// TwinCAT 3 PLC project Hammerschmied
// ProgramVersion: 3.1.4023.0
// libraries:
//   EfficientIO Communicator, * (EfficientIO)
//   EfficientIO Energy Basic, * (EfficientIO)
//   EfficientIO ModbusTCP, * (EfficientIO)
//   Lynus Persistent Data V1, * (Lynus AG)
//   Lynus Standards, * (EfficientIO)
//   Tc2_Standard, * (Beckhoff Automation GmbH)
//   Tc2_System, * (Beckhoff Automation GmbH)
//   Tc2_Utilities, * (Beckhoff Automation GmbH)
//   Tc3_Module, * (Beckhoff Automation GmbH)
// project tree:
//   / FastTask.TcTTO (not stored), MiddleTask.TcTTO, SlowTask.TcTTO
//   FB/ FB_EMS_T.TcPOU (excluded from build), FB_EMS_V12.TcPOU, FB_EM_Beckhoff_KL3403.TcPOU (not stored), FB_IntervalBit.TcPOU (not stored)
//   POUs/ prgBattery.TcPOU, prgComEffIO.TcPOU, prgCS.TcPOU, prgEM.TcPOU, prgEMS.TcPOU, prgGrid.TcPOU, prgHouse.TcPOU, prgPersistent.TcPOU (not stored), prgPV.TcPOU, prgRWEffIO.TcPOU, prgVarEffIO.TcPOU (not stored)
// real-time tasks:
//   TASK FastTask: cycle T#5ms, priority 6, ADS port 350
//   TASK MiddleTask: cycle T#10ms, priority 8, ADS port 351
//   TASK SlowTask: cycle T#20ms, priority 10, ADS port 352
// I/O:
//   DEVICE Gerät 2 (CX-BK)
//     Box 1 (CX-BK)
// variable links:
//   Hammerschmied/Hammerschmied Instance <-> Device 2 (CX-BK)/Box 1 (CX-BK)
//     MiddleTask Inputs/prgEM.fbEM1.fbKL3403.byStateCH1 <-> Term 2 (KL3403)/Channel 1/Status
//     MiddleTask Inputs/prgEM.fbEM1.fbKL3403.byStateCH2 <-> Term 2 (KL3403)/Channel 2/Status
//     MiddleTask Inputs/prgEM.fbEM1.fbKL3403.byStateCH3 <-> Term 2 (KL3403)/Channel 3/Status
//     MiddleTask Inputs/prgEM.fbEM1.fbKL3403.iDataInCH1 <-> Term 2 (KL3403)/Channel 1/Daten Ein
//     MiddleTask Inputs/prgEM.fbEM1.fbKL3403.iDataInCH2 <-> Term 2 (KL3403)/Channel 2/Daten Ein
//     MiddleTask Inputs/prgEM.fbEM1.fbKL3403.iDataInCH3 <-> Term 2 (KL3403)/Channel 3/Daten Ein
//     MiddleTask Inputs/prgEM.fbKBusState.uiKBusState_OUT <-> Inputs/State
//     MiddleTask Outputs/prgEM.fbEM1.fbKL3403.byCntrCH1 <-> Term 2 (KL3403)/Channel 1/Kontrolle
//     MiddleTask Outputs/prgEM.fbEM1.fbKL3403.byCntrCH2 <-> Term 2 (KL3403)/Channel 2/Kontrolle
//     MiddleTask Outputs/prgEM.fbEM1.fbKL3403.byCntrCH3 <-> Term 2 (KL3403)/Channel 3/Kontrolle

CONFIGURATION Hammerschmied
    RESOURCE PLC ON TwinCAT3
        TASK MiddleTask(INTERVAL := T#10ms, PRIORITY := 8);
        TASK SlowTask(INTERVAL := T#20ms, PRIORITY := 10);
        PROGRAM prgBattery WITH MiddleTask : prgBattery;
        PROGRAM prgCS WITH MiddleTask : prgCS;
        PROGRAM prgEMS WITH MiddleTask : prgEMS;
        PROGRAM prgGrid WITH MiddleTask : prgGrid;
        PROGRAM prgHouse WITH MiddleTask : prgHouse;
        PROGRAM prgPersistent WITH MiddleTask : prgPersistent;
        PROGRAM prgPV WITH MiddleTask : prgPV;
        PROGRAM prgEM WITH MiddleTask : prgEM;
        PROGRAM prgComEffIO WITH SlowTask : prgComEffIO;
    END_RESOURCE
END_CONFIGURATION

// ---- POUs/prgBattery.TcPOU
PROGRAM prgBattery
VAR PERSISTENT
	bEnableBattery				: BOOL;							//{#lynus.ag#()}
	byPrioBattery				: BYTE;							//{#lynus.ag#()}
	lrMaxCapacityBattery		: LREAL;						//{#lynus.ag#()}
	lrCounterBattProd			: LREAL;						//{#lynus.ag#()}
	lrCounterBattCons			: LREAL;						//{#lynus.ag#()}
	by_Min_BatterySOC			: BYTE;							//{#lynus.ag#()}
	by_Max_BatterySOC			: BYTE;							//{#lynus.ag#()}
END_VAR
VAR
	fbBattery					: FB_Xelectrix_Powerbox_v2_2;
	fbBattCounter				: FB_EnergyCounter;
	bIsEnabledBattery			: BOOL;							//{#lynus.ag#()}
	bResetBattery				: BOOL;							//{#lynus.ag#()}
	bSResetBattery				: BOOL;							//{#lynus.ag#()}
	byErrorWarningBattery		: BYTE;							//{#lynus.ag#()}
	dwSOCBattery				: DWORD;						//{#lynus.ag#()}
	rTargetPowerBattery			: REAL;							//{#lynus.ag#()}
	lrPowerBattery				: LREAL;						//{#lynus.ag#()}
	lrActualCapacityBattery		: LREAL;						//{#lynus.ag#()}
	mtest: BOOL;

	int_GridState: INT;											//{#lynus.ag#()}
	int_BatteryState: INT;										//{#lynus.ag#()}
	int_OperatingState: INT;									//{#lynus.ag#()}
	int_ErrorState: INT;										//{#lynus.ag#()}

	FB_Interval: FB_IntervalBit;
	m_IslandOperationStart: BOOL;								//{#lynus.ag#()}
	m_IslandOperationOngoing: BOOL;								//{#lynus.ag#()}
	m_IslandOperationStop: BOOL;								//{#lynus.ag#()}
	t_Interval :TIME:=T#30M;
	t_HightTime :TIME:=T#1S;
	
	m_BatteryErrorActive: BOOL;									//{#lynus.ag#()}
	m_BatteryModbusCommError: BOOL;								//{#lynus.ag#()}
	m_BatteryTargetSPError: BOOL;								//{#lynus.ag#()}
	Ton_Delay_BatteryError: Ton;
	Ton_Delay_BatteryModbusError: Ton;
	Ton_Delay_BatterySPError: Ton;	
	by_S_Min_BatterySOC			: BYTE;							//{#lynus.ag#()}
	by_S_Max_BatterySOC			: BYTE;							//{#lynus.ag#()}
	
END_VAR


IF mtest THEN
	Lynus_Standards.GVL_Energy.stDataOfBatteryInverters[1,1].rTargetPowerEMS:=0;
	mtest:=FALSE;
 END_IF
 
 
 
fbBattery(
	bEnable:= bEnableBattery, 
	bActivateControl:= TRUE, 
	byUnitID:= 1, 
	byPriority:= byPrioBattery, 
	diNrOfEMS_IN:= prgEMS.fbEMS.diNrOfEMS_OUT, 
	lrMaxCapacityBattery:= lrMaxCapacityBattery, 
	sIPAdress:= '192.168.1.235', 						// modify IP Adress
	bReset:= bResetBattery, 
	by_minDischargeSOC := by_Min_BatterySOC,
	by_maxChargeSOC := by_Max_BatterySOC,
	stDataXelectrix=> , 
	stDataBatt=> , 
	stDataBattInverter=> , 
	stDataEMPower_Grid=> , 
	stDataEMCounter_Grid=> , 
	diNrOfBatt_OUT=> , 
	diNrOfBattInverter_OUT=> , 
	diNrOfEM_OUT_Grid=> , 
	lrMaxCapacityBattery_OUT=> ,	
	by_SminDischargeSOC	=> by_S_Min_BatterySOC,	
	by_SmaxChargeSOC=> by_S_Max_BatterySOC
);
	
//Out
bIsEnabledBattery := fbBattery.stDataBatt.bEnabled;
	bSResetBattery := fbBattery.stDataBattInverter.bStateReset;
		dwSOCBattery := fbBattery.stDataBatt.dwSOC;
			rTargetPowerBattery := fbBattery.stDataBattInverter.rTargetPower;
				lrPowerBattery := fbBattery.stDataBatt.lrPower;
					lrActualCapacityBattery := fbBattery.lrMaxCapacityBattery_OUT;	
						byErrorWarningBattery := fbBattery.stDataBatt.byErrorWarning;
						
						
// EnergyCounter
fbBattCounter(
	byActiveTariff:= 1, 
	lrPowerInput:= lrPowerBattery, 
	lrTotalCounterEnergy_Consumption=> , 
	lrTotalCounterEnergy_Production=> , 
	lrCounterEnergyT1_Consumption=> , 
	lrCounterEnergyT2_Consumption=> , 
	lrCounterEnergyT1_Production=> , 
	lrCounterEnergyT2_Production=> );
	
IF fbBattCounter.lrTotalCounterEnergy_Production > lrCounterBattProd THEN  	
	lrCounterBattProd := fbBattCounter.lrTotalCounterEnergy_Production;
END_IF

IF fbBattCounter.lrTotalCounterEnergy_Consumption > lrCounterBattCons THEN  	
	lrCounterBattCons := fbBattCounter.lrTotalCounterEnergy_Consumption;
END_IF

// send e states to cloud
int_GridState 		:= fbBattery.stDataXelectrix.eGridState;
int_BatteryState	:= fbBattery.stDataXelectrix.eBatteryState;
int_OperatingState	:= fbBattery.stDataXelectrix.eOperatingState;
int_ErrorState		:= fbBattery.stDataXelectrix.eErrorState;


// create bits when battery is in island operation

FB_Interval(
	m_Input			:=  prgBattery.fbBattery.stDataXelectrix.eGridState = 2,	//   2 = Island Mode 
	t_Interval 		:= t_Interval , 
	t_HighTime		:= t_HightTime, 
	m_RisingEdge	=> m_IslandOperationStart, 
	m_Interval		=> m_IslandOperationOngoing, 
	m_FallingEdge	=> m_IslandOperationStop);

// monitoring Battery status

Ton_Delay_BatteryError (In := fbBattery.stDataXelectrix.eErrorState =2,
						PT :=T#5S,
						Q => m_BatteryErrorActive);

Ton_Delay_BatteryModbusError (	In := fbBattery.stDataXelectrix.eErrorState = 1,
								PT :=T#10M,
								Q => m_BatteryModbusCommError);						

Ton_Delay_BatterySPError (	In := ABS(fbBattery.iSetpointPower/10-lrPowerBattery) > 20 AND fbBattery.stDataXelectrix.eGridState<>2 AND fbBattery.stDataBatt.dwSOC<90,	// not alarming during island operation
							PT :=T#1M,
							Q => m_BatteryTargetSPError);

END_PROGRAM

// ---- POUs/prgEMS.TcPOU
PROGRAM prgEMS
VAR PERSISTENT
	byMaxDepthOfDischrgEPO		: BYTE;							//{#lynus.ag#()}
	byPrioMinChrgBattSOCInEPO	: BYTE;							//{#lynus.ag#()}
	byResChrgfromGridToBatt		: BYTE;							//{#lynus.ag#()}
	byReserveSOCEPO				: BYTE;							//{#lynus.ag#()}
	uiUpdateTime				: UINT;							//{#lynus.ag#()}
	bEnableEMS					: BOOL;							//{#lynus.ag#()}
	bAllowChrgFromGrid			: BOOL;							//{#lynus.ag#()}
	rMainFuseCSEMS				: REAL;							//{#lynus.ag#()}
	iOperationModeEMS			: INT;							//{#lynus.ag#()}
	by_MinSOC_AdaptiveLC		: BYTE;							//{#lynus.ag#()}
END_VAR
VAR
	fbEMS						: FB_EMS_V12;
	bIsEnableEMS				: BOOL;							//{#lynus.ag#()}
	bStateAllowChrgFromGrid		: BOOL;							//{#lynus.ag#()}
	bHPActivate					: BOOL;							//{#lynus.ag#()}
	bControllingState			: BOOL;							//{#lynus.ag#()}
	iMessageEMS					: INT;							//{#lynus.ag#()}
	rHeartbeatEMS				: REAL;							//{#lynus.ag#()}
	rErrorWarningEMS			: REAL;							//{#lynus.ag#()}
	rReadyEMS					: REAL;							//{#lynus.ag#()}
	rNewBatteryPowerEMS			: REAL;							//{#lynus.ag#()}
	b_EnableBatteryChargingControl				: BOOL:=TRUE;							//{#lynus.ag#()}
	b_StartReleaseBatteryCharging				: BOOL;									//{#lynus.ag#()}
	b_StopReleaseBatteryCharging				: BOOL;									//{#lynus.ag#()}
	b_TimeBasedReleaseChargingBattery			: BOOL;									//{#lynus.ag#()}
	b_StartManualCharging						: BOOL;									//{#lynus.ag#()}
	b_StartManualCharging_SOC					: BOOL;									//{#lynus.ag#()}
	r_Charging_SOC_SetPoint						: REAL;									//{#lynus.ag#()}
	RS_ManualCharging: Rs;
	RS_ManualCharging_SOC: Rs;
	TON_ManualCharging: Ton;
	time_ManualCharging: TIME:=T#2H;
	r_trig_ManualCharging: R_trig;
	f_trig_ManualCharging: f_trig;
	r_trig_ManualCharging_SOC: R_trig;
	f_trig_ManualCharging_SOC: f_trig;
	r_trig_b_StartManualCharging: R_trig;
	r_trig_b_StartManualCharging_SOC: R_trig;
	m_test: BOOL;
	b_dummy						: bool;									//{#lynus.ag#()}
	iOperationModeEMS_actual			: INT;							//{#lynus.ag#()}

	mtest: BOOL;
	m_Enable_Dynamic_LM: BOOL;
END_VAR

fbEMS.stSetupEMS.bAllowChrgFromGrid := bAllowChrgFromGrid or RS_ManualCharging.Q1;
fbEMS.stSetupEMS.byMaxDepthOfDischrgEPO := byMaxDepthOfDischrgEPO;
fbEMS.stSetupEMS.byPrioMinChrgBattSOCInEPO := byPrioMinChrgBattSOCInEPO;
fbEMS.stSetupEMS.byResChrgfromGridToBatt := byResChrgfromGridToBatt;
fbEMS.stSetupEMS.byReserveSOCEPO := byReserveSOCEPO;
fbEMS.stSetupEMS.rSizeMainFuseCS := rMainFuseCSEMS;
fbEMS.stSetupEMS.uiUpdateTime := uiUpdateTime;
(*IF m_Enable_Dynamic_LM THEN
	IF prgBattery.dwSOCBattery > byMinSOCdynamicLM AND NOT prgCS.bCarConnected THEN
		iOperationModeEMS := 1;
	ELSE
		iOperationModeEMS := 3;
	END_IF  
END_IF

IF iOperationModeEMS = 0 THEN fbEMS.eOperationMode := E_OperatingMode_EMS.eAllOff;
ELSIF iOperationModeEMS = 1 THEN fbEMS.eOperationMode := E_OperatingMode_EMS.eSelfConsumption;	
ELSIF iOperationModeEMS = 2 THEN fbEMS.eOperationMode := E_OperatingMode_EMS.ePeakLoadCapping;
ELSIF iOperationModeEMS = 3 THEN fbEMS.eOperationMode := E_OperatingMode_EMS.eLoadManagement;			
END_IF
*)
IF iOperationModeEMS = 0 THEN 
	fbEMS.eOperationMode_Ext := E_OperatingMode_EMS.eAllOff;
ELSIF iOperationModeEMS = 1 THEN 
	fbEMS.eOperationMode_Ext := E_OperatingMode_EMS.eSelfConsumption;	
ELSIF iOperationModeEMS = 2 THEN 
	fbEMS.eOperationMode_Ext := E_OperatingMode_EMS.ePeakLoadCapping;
ELSIF iOperationModeEMS = 3 THEN 
	fbEMS.eOperationMode_Ext := E_OperatingMode_EMS.eLoadManagement;			
ELSIF iOperationModeEMS = 4 THEN 
	fbEMS.eOperationMode_Ext := E_OperatingMode_EMS.eAdaptiveLoadControl;		
END_IF

fbEMS(
	bEnable:= bEnableEMS, 
	diNrOfEM_IN_ECS:= , 
	stSetupEMS:= , 
	eOperationMode_Ext:= , 
	eSpeedModeBackendController:= E_SpeedModeBackendController_EMS.eSlow,	//.efast, 
	eSpeedModeLocalController:= E_SpeedModeLocalController_EMS.eSlow,    //efast,
	bZeroPowerRegulation	:= FALSE, 
	b_EnableBatteryChargingControl	:= b_EnableBatteryChargingControl,
	b_StartReleaseBatteryCharging 	:= b_StartReleaseBatteryCharging OR r_trig_ManualCharging.Q ,
	b_StopReleaseBatteryCharging 	:= b_StopReleaseBatteryCharging OR (f_trig_ManualCharging.Q AND NOT b_StartReleaseBatteryCharging) OR (f_trig_ManualCharging_SOC.Q AND NOT b_StartReleaseBatteryCharging) ,
	by_MinSOC_AdaptiveLC:= by_MinSOC_AdaptiveLC, 
	bActivateHP:= bHPActivate, 
	bControllingState:= TRUE, //bControllingState, 
	rHeartbeat:= rHeartbeatEMS, 
	rErrorWarning:= rErrorWarningEMS, 
	rEnergyOptReady:= rReadyEMS, 
	rNewBattPower:= rNewBatteryPowerEMS,
	b_AnyCarConnected:= prgCS.bCarConnected , 
	rMaxBattChargingPower:= , 
	rPeakDetectionforCalculation:= , 
	eMessageEMS=> iMessageEMS, 
	bStateEnable=> bIsEnableEMS, 
	bStateAllowChrgFromGrid=> bStateAllowChrgFromGrid, 
	bMissingPowerData=> , 
	bSurplusAvailable=> , 
	byProgress=> , 
	uiState_OUT=> , 
	diNrOfEMS_OUT=> , 
	arrMinPrioReached=> , 
	arrMaxPrioReached=> , 
	b_TimeBasedReleaseChargingBattery => b_TimeBasedReleaseChargingBattery);

iOperationModeEMS_actual := fbEMS.eOperationMode;

(*
fbEMS(
	bEnable:= bEnableEMS, 
	diNrOfEM_IN_ECS:= , 
	stSetupEMS:= , 
	eOperationMode:= , 
	eSpeedModeBackendController:= E_SpeedModeBackendController_EMS.efast, 
	eSpeedModeLocalController:= E_SpeedModeLocalController_EMS.efast,
	bActivateHP:= bHPActivate, 
	bControllingState:= TRUE, //bControllingState, 
	rHeartbeat:= rHeartbeatEMS, 
	rErrorWarning:= rErrorWarningEMS, 
	rEnergyOptReady:= rReadyEMS, 
	rNewBattPower:= rNewBatteryPowerEMS, 
	b_ZeroPowerRegulation	:= FALSE,
	b_EnableBatteryChargingControl	:= b_EnableBatteryChargingControl,
	b_StartReleaseBatteryCharging 	:= b_StartReleaseBatteryCharging OR r_trig_ManualCharging.Q ,
	b_StopReleaseBatteryCharging 	:= b_StopReleaseBatteryCharging OR (f_trig_ManualCharging.Q AND NOT b_StartReleaseBatteryCharging) OR (f_trig_ManualCharging_SOC.Q AND NOT b_StartReleaseBatteryCharging) ,
	rMaxBattChargingPower			:= ,
	rPeakDetectionforCalculation	:=,
	eMessageEMS=> iMessageEMS, 
	bStateEnable=> bIsEnableEMS, 
	bStateAllowChrgFromGrid=> bStateAllowChrgFromGrid, 
	bMissingPowerData=> , 
	bSurplusAvailable=> , 
	byProgress=> , 
	uiState_OUT=> , 
	diNrOfEMS_OUT=> , 
	arrMinPrioReached=> , 
	arrMaxPrioReached=> ,
	b_TimeBasedReleaseChargingBattery => b_TimeBasedReleaseChargingBattery);
*)
	
// code for manual charging button, time hardcoded to 2h with variable 	time_ManualCharging
	
r_trig_b_StartManualCharging(clk:=b_StartManualCharging);
r_trig_b_StartManualCharging_SOC(clk:=b_StartManualCharging_SOC);
RS_ManualCharging_SOC(	Set := r_trig_b_StartManualCharging_SOC.Q AND NOT RS_ManualCharging_SOC.Q1 AND REAL_TO_DWORD(r_Charging_SOC_SetPoint) > prgBattery.dwSOCBattery AND NOT b_TimeBasedReleaseChargingBattery AND NOT RS_ManualCharging.Q1,
						Reset1 := (r_trig_b_StartManualCharging_SOC.Q AND RS_ManualCharging_SOC.Q1) OR REAL_TO_DWORD(r_Charging_SOC_SetPoint) <= prgBattery.dwSOCBattery OR b_StartReleaseBatteryCharging);
IF 	(r_trig_b_StartManualCharging.Q OR r_trig_b_StartManualCharging_SOC.Q) AND NOT b_TimeBasedReleaseChargingBattery AND NOT RS_ManualCharging.Q1 THEN
	RS_ManualCharging.SET:=TRUE;
ELSIF (r_trig_b_StartManualCharging.Q  AND RS_ManualCharging.Q1) OR (TON_ManualCharging.Q AND NOT RS_ManualCharging_SOC.Q1)  OR b_StartReleaseBatteryCharging OR f_trig_ManualCharging_SOC.Q THEN
	RS_ManualCharging.RESET1:=TRUE;		
END_IF
TON_ManualCharging(	In:=RS_ManualCharging.Q1, PT:= time_ManualCharging);

RS_ManualCharging();
RS_ManualCharging.SET:=FALSE;
RS_ManualCharging.RESET1:=FALSE;
r_trig_ManualCharging(clk:=RS_ManualCharging.Q1);
f_trig_ManualCharging(clk:=RS_ManualCharging.Q1);
r_trig_ManualCharging_SOC(clk:=RS_ManualCharging_SOC.Q1);
f_trig_ManualCharging_SOC(clk:=RS_ManualCharging_SOC.Q1);

			
// Test
IF REAL_TO_DWORD(r_Charging_SOC_SetPoint) > prgBattery.dwSOCBattery  THEN
	mtest := TRUE;
ELSE
	mtest := FALSE;
END_IF

END_PROGRAM

// ---- FB/FB_EMS_V12.TcPOU
FUNCTION_BLOCK FB_EMS_V12
VAR_INPUT PERSISTENT
	bEnable										: BOOL;																								//{#lynus.ag#()} //Enable and dissable this function
	diNrOfEM_IN_ECS								: DINT;																								//Number of the electric meter for incoming power data. (Its for the complete consumption of all charging stations)
	stSetupEMS									: ST_Setup_EMS := (uiUpdateTime := 15);																//{#lynus.ag#()} //Setup EMS
	eOperationMode_Ext							: E_OperatingMode_EMS;																				//{#lynus.ag#()} //Operation Mode EMS
	eSpeedModeBackendController					: E_SpeedModeBackendController_EMS;																	//Speed for the Controller what discharge the Battery when the commands come from the Backend
	eSpeedModeLocalController					: E_SpeedModeLocalController_EMS;																	//Speed for the local Controller for charge and discharge the Battery
	bZeroPowerRegulation						: BOOL;																								//{#lynus.ag#()} // activates the Battery discharging before using the mains during LoadManagement; Line 1728/1732/1738
	b_EnableBatteryChargingControl				: BOOL;																								//{#lynus.ag#()} //  
	b_StartReleaseBatteryCharging				: BOOL;																								//{#lynus.ag#()} //  
	b_StopReleaseBatteryCharging				: BOOL;																								//{#lynus.ag#()} //  
	by_MinSOC_AdaptiveLC						: BYTE; 
END_VAR
VAR_INPUT
	bActivateHP									: BOOL;																								//{#lynus.ag#()} //Activate the Heating pumps when the Backend deliver the signal. NOT OVERRIDE
	bControllingState							: BOOL;																								//{#lynus.ag#()} //The control state of the service is linked here. NOT OVERRIDE
	rHeartbeat									: REAL;																								//{#lynus.ag#()} //Heartbeat from the Service. NOT OVERRIDE
	rErrorWarning								: REAL;																								//{#lynus.ag#()} //Error or Warning from the Service. NOT OVERRIDE
	rEnergyOptReady								: REAL;																								//{#lynus.ag#()} //Energy Optimization Service Ready. NOT OVERRIDE
	rNewBattPower								: REAL;																								//{#lynus.ag#()} //New Battery Power from Backend Service. NOT OVERRIDE
	b_AnyCarConnected							: BOOL;																								// requrired for the dadaptive load control 
	rMaxBattChargingPower						: REAL:=100;																								// Maximum Battery Charging power in percent
	rPeakDetectionforCalculation				: REAL:=3;																								// Value for Peak detection, was original 3 but caused issues with fast changing loads (e.g. industrie)
END_VAR
VAR_OUTPUT
	eMessageEMS									: Lynus_Standards.E_Message_EMS;																	//EMS Message
	bStateEnable								: BOOL;																								//{#lynus.ag#()} //Show if the ems function is enabled or not
	bStateAllowChrgFromGrid						: BOOL;																								//{#lynus.ag#()} //Show the State if the charging from grid is allowed or not
	bMissingPowerData							: BOOL;																								//Missing data on the max power setup from one ore more devices
	bSurplusAvailable							: BOOL;																								//Variable that indicates if there is surplus or not
	byProgress									: BYTE;																								//Shows the Progress from the new Calculation when we have Surplus. When we have no Surplus and we discharge the batterys this Value is on 100
	uiState_OUT									: UINT;																								//Actual State
	diNrOfEMS_OUT								: DINT;																								//Active Number from the EMS Function for using on other functions
	arrMinPrioReached							: ARRAY[1..5] OF BOOL;																				//Shows if all different devices types are set to 0% with the target power ([1] = Battery, [2] = HP, [3] = EHE, [4] = OBC, [5] = ECS)
	arrMaxPrioReached							: ARRAY[1..5] OF BOOL;																				//Shows if all different devices types are set to 100% with the target power ([1] = Battery, [2] = HP, [3] = EHE, [4] = OBC, [5] = ECS)	
	b_TimeBasedReleaseChargingBattery			: BOOL;																								//
END_VAR	
VAR
	eOperationMode								: E_OperatingMode_EMS;																				//{#lynus.ag#()} //Operation Mode EMS
	(*-----------------------------------------------------------------------Internal Variables and Functions for connection to the Backend--------------------------------------------------------------------------------*)
	fbPIDDischrgCmdFromBackend					: FB_PID;																							//PID Contrller what controll the discharging power from the Battery when the controlling from backend is activated
	timDissableFunctions						: TON;																								//Timer to dissable the Function after Lynus_Standards.Constants_General.tTimeDissableLynusFunctions Days without connection to the Lynus Cloud
	timResetConnectionOnGVL						: TON;																								//Timer to try reset the connection Flag on the GVL. (When somebody delete the Connection Function and make only a onlinechange)
	timHB										: TON;																								//Timer to check the Heartbeat from the Backendservice
	timPIDDischrgCmdFromBackend					: TON;																								//Timer to set the output from the pid controller to 0 due to internal control deviations (Backend Mode)
	timCorrectionSetpoint						: TOF;																								//Timer to make the correction on the Setpoint for Battery power. This is neccessary to give time to the inverter and Grid to adjust on the new values
	timErrorWarning								: TON;																								//Timer to enable the Function Backend Mode after a Error or Warning
	timEnergyOptReady							: TON;																								//Timer to enable the Function Backend Mode after the Backend Service is ready
	timControlingState							: TON;																								//Timer to enable the controlling over the Backend Mode
	timResetActivateHP							: TON;																								//Timer to reset the Activate HP Command from the Backend Service
	FPEnablePID									: R_TRIG;																							//Internal positive edge
	FPMakeCorrection							: R_TRIG;																							//Internal positive edge
	bDischrgCmdFromBackendOK					: BOOL;																								//Allowed to controll the Devices from Backend
	rHeartbeat_CP								: REAL;																								//Compare the Heartbeat from the Backend
	rControllerQPIDDischrgCmdFromBackend		: REAL;																								//Controller output from pid controll over Backend Mode
	rNewBattPower_CP							: REAL;																								//New Battery power to ckeck if we have received a new Value in kW
	lrActualPowerBatterys						: LREAL;																							//Actual Power from the Batterys in kW
	lrErrorPIDCorrectionDischrgCmdFromBackend	: LREAL;																							//Limit the Error on the pid controller for discahrge the battery on the controll over Backend Mode
	lrNewBatteryPowerWithCorrection				: LREAL;																							//The New Battery power from the Backend with correction that we dont insert power in the Grid
	liLPDischrgCmdFromBackend					: LINT;																								//Loop to send the command from Backend to the Devices
	(*-----------------------------------------------------------------------------------Rest of internal Variabels and Functions---------------------------------------------------------------------------------------*)
	fbMessagesEMS								: FB_EMS_Message;																					//FB to create the Messages for this Function
	fbNumberDevice								: FB_NumberOfDevice;																				//Function block to calcualte the number of the Device
	fbTaskIndex									: GETCURTASKINDEX;																					//Function to read out the Task Index in witch the function is running
	fbPIDBatterySC								: FB_PID;																							//PID Controller to discharge the battery in the self consumption mode
	fbPIDBatteryEPO								: FB_PID;																							//PID Controller to discharge the battery in the emergency power mode
	fbPIDBatteryPLCLM_Dischrg					: FB_PID;																							//PID Controller to Dischage the battery on load management mode and peak shaving mode
	fbPIDBatteryPLCLM_Chrg						: FB_PID;																							//PID Controller to Charge the battery on load management mode and peak shaving mode
	timCalculateNewPowerValue					: TON;																								//Timer to start a new session to calculate the new power value for the devices
	timPIDSC									: TON;																								//Timer to set the output from the pid controller to 0 due to internal control deviations (Self consumption mode)
	timPIDEPO									: TON;																								//Timer to set the output from the pid controller to 0 due to internal control deviations (Emergency power mode)
	timCorrectionECS							: TON;																								//Timer for make the correction for ECS in the Load management and peak capping mode with use the separate fuse
	timErrorGridMessurement						: TON;																								//Timer with delay to stop the EMS Function if we have a error on the Grid messurement
	timTimeout									: TON;																								//Timer for Timout
	timCutPeaks									: TOF;																								//Timer to cut peaks on the grid. The system waits for this time for strong and short peaks before regulating.
	timDelayStart								: TOF;																								//Timer with the delay to start the ems function after a online change
	timResetDisableECS							: TOF;																								//Timer to reset the dissbling the ECS after a Error from the Electric Meter what messure the power from all ECS
	FPEPO										: R_TRIG;																							//Internal positive edge
	FNEPO										: F_TRIG;																							//Internal negative edge
	eOperationModeEMS_CP						: E_OperatingMode_EMS;																				//Operation Mode EMS/Battery to compare with the original variable
	arrPD										: ARRAY[1..12] OF FB_PersistentData_Number;															//Function to save persistent data
	arrTimBatterysAreFull						: ARRAY[1..Constants_Energy.diMaxNumberOfBatteryInverters] OF TON;									//Timer start for each Battery when is full
	arrActualStepInTurn_CP						: ARRAY[1..2] OF BYTE;																				//Actual Step in turn to compare with original variable
	arrActualPrioInTurn							: ARRAY[1..5] OF BYTE;																				//Actual Priority (1-255) that is currently in turn ([1] = Battery, [2] = HP, [3] = EHE, [4] = OBC, [5] = ECS)
	arrActualStepInTurn							: ARRAY[1..2] OF BYTE;																				//Actual Step (1-10) from step switched devices that is currently in turn ([1] = HP, [2] = EHE)
	arrLPPrioZeroSetToZeroP						: ARRAY[1..5] OF LINT;																				//Array with loop to set each device with priority 0 to the target power value 
	arrCTCheckActivePrio						: ARRAY[1..5] OF LINT;																				//Array with loop to check the actual prioritys
	bEPMActive									: BOOL;																								//Emergency power mode is active
	bChargePrioBatterysOnEPO					: BOOL;																								//Load batterys that made a island grid first to the adjustable SOC before start with al other devices
	bStepWasOn100								: BOOL;																								//Its true when the actual step from step switched devices was on 100%
	bECSPrio255									: BOOL;																								//True when we reached the max prio of the charging stations
	bStopAll									: BOOL;																								//Stop the EMS when we some is happend what make trouble
	bDisableECS									: BOOL;																								//Dissable the ECS when the EM what messure the power from all ECS has a error
	bErrorOnGridMessurement						: BOOL;																								//Shows if on the Grid Messurement is a error and stop then the EMS Function
	bNoPowerForECS								: BOOL;																								//Variable what shows that we dont can give more power on the ECS because we have to much power on the Fuse line on wich the ECS is connected
	bySmGrActiveCommonPrio_CP					: BYTE;																								//Smalest or greatest active common priority of the devices to compare with the original varible
	byLPSmActiveCommonPrio						: BYTE;																								//Loop to check the smalest active common priority
	bySmGrActiveCommonPrio						: BYTE;																								//Smalest or greatest active common priority of the devices
	bySearchBigestPrio							: BYTE;																								//Search the biggest Prio for each device in the Steps in what we choose the prio
	uiState										: UINT;																								//Actual State
	uiState_CP									: UINT;																								//Actual State to compare for activating the timout timer
	diNumberOfDevicesFromEachType				: DINT;																								//Count the Number of each Device what has a priority <> 0
	diMemCmpOperationState						: DINT;																								//Variable to compare the operation state			
	diNumberOfActiveBatterys					: DINT;																								//Number of active batterys
	diNumberOfBatteryInverterInEPO				: DINT;																								//Number of battery inverters that work in Emergency Power operation 
	diNrOfEM_IN_CS_CP							: DINT;																								//Number of the electric meter for receive data. (Its for the complete consumption of all charging stations to compare)
	diNumberOfECS								: DINT;																								//Number of total charging stations on what the power must reduced with the max fuse power
	diBiggestNumberOfDeviceConstants			: DINT;																								//Biggest Number of the constants for the several device types. Needs to calcualte the delay for the timout timer
	dwSumSOC									: DWORD;																							//Sum of the SOC from all batterys
	dwSumSOCInEPO								: DWORD;																							//Sum of the SOC from all batterys that make a island mode at the moment
	dwAvarageBatterySOC							: DWORD;																							//Actual avarage Battery SOC from each Battery
	dwAvarageBatterySOCInEPO					: DWORD;																							//Actual avarage Battery SOC from each Battery that make a island mode at the moment
	udiCounterOnlineChange_CP					: UDINT;																							//Counter for online change to comapre it	
	udiCycleTime								: UDINT;																							//Cycle time in wich the function is running. Needs to calculate the delay for the timout timer
	rValuePercentToControllableDevices			: REAL;																								//Percent value to set the target power to controllable devices
	rValuePercentToStepSwitchedDevices			: REAL;																								//Percent value to set the target power to on/off or step switched devices
	rControllerQPIDSC							: REAL;																								//Controller output from pid self consumption
	rControllerQPIDEPO							: REAL;																								//Controller output from pid emergency power operation
	rSizeMainFuseCS_CP							: REAL;																								//Size of the main fuse form the charging stations to compare with the original varialbe
	lrTargetPowerCorrectionECS					: LREAL;																							//New Target power for chargign station after correction with max fuse power
	lrPowerDiffFuseECS							: LREAL;																							//Power difference between max fuse power charging station and actual power for all charging stations 
	lrPowerForCalculateECS						: LREAL;																							//Power to calcualte the % for each charging station
	lrGridPower									: LREAL;																							//Grid power in kW
	lrGridPower_CP								: LREAL;																							//Grid power in kW to compare for correction when the backend is controlling the battery
	lrSizeBatteryPowerInEPO						: LREAL;																							//Power in kW of all Battery inverters that are made a island mode at the moment
	lrSizeGridConnection						: LREAL;																							//Size of the complete grid connection
	lrActualSurplusOrConsumption				: LREAL;																							//Actual surplus or consumption in kW
	lrActualSurplusOrConsumptionOld				: LREAL;																							//Old value from last step with surplus or consumption in kW
	lrMaxPowerDevicesWithActualPrio				: LREAL;																							//Actual complete max power from all devices with the same priority
	lrErrorPIDCorrectionBattSC					: LREAL;																							//Limit the Error on the pid controller for discahrge the battery on the self consumption mode
	lrErrorPIDCorrectionBattEPO					: LREAL;																							//Limit the Error on the pid controller for discahrge the battery on the emergency power operation mode
	lrErrorPIDCorrectionBattPLCLM_Dischrg		: LREAL;																							//Limit the Error on the pid controller for discahrge the battery on the load management mode and peak shaving mode
	lrErrorPIDCorrectionBattPLCLM_Chrg			: LREAL;																							//Limit the Error on the pid controller for charge the battery on the load management mode and peak shaving mode
	liCounterCkeckDeviceAndPrio					: LINT;																								//Counter to ckeck the device and Prio in the Steps for HP and EHE. Here we didn't can use a loop regarding performance problems on small PLC
	liNrOfNotDoneDevices						: LINT;																								//Shows the Numer of Devices what are not controlled with the minimum or the maximum power when we have a actual Prio from 1 or 255. That we can set the min reached or max reached Flag
	liLPCheckDeviceAndPrio						: LINT;																								//Loop to ckeck the Number of Devices and the Prio
	liLPGridData								: LINT;																								//Loop to check some grid data
	liLPActualSurplusOrConsumption				: LINT;																								//Loop to check actual surplus or consumption
	liLPBatterysSetupData						: LINT;																								//Loop to copy the setup data from the battery inverters
	liLPBatteryData								: LINT;																								//Loop to check some data from batterys
	liLPSumSOCInEPO								: LINT;																								//Loop to calculate the sum of the SOC from all batterys that buils a island mode at the moment
	liLPInEPO									: LINT;																								//Loop to check if 1 or more battery inverters build a island grid
	liLPCheckMaxPower							: LINT;																								//Loop to ckeck the max power from each device
	liLPSetPercentPower							: LINT;																								//Loop to set the calculatet percetn power to the device
	liLPCorrectionPowerCS						: LINT;																								//Loop to make a correction on the target power from the charging stations in dependence of the max fuse power 
	liLPDataBatteryInverter						: LINT;																								//Loop to check or set data from battery inverters
	RS_BatteryChargingControl: RS;
END_VAR

//Creator : Stefan Lackner
//Company : EfficientIO
//Date : 20.03.2024
//Version : 1.2.0.0
//With this FB the EMS control can be realized on the PLC. 
//This divides the excess energy among the devices according to priority
//Devices with priority 0 received as target power 0
//If we have less or no surplus, then the target power will be reduced or remains on the same value
//The EMS function can handle batterie devices, controllable devices, On/Off devices and step switched devices. 
//If we have no surplus, and all devices has a target power from 0, then the battery try to balancing the consumption.
//This depends what operation mode is active
//If the mode load managemant is active, for the charging station the max power from the fuse is neccessary, because the ems dont can use all the power from the max. grid power for the charging stations.  
//When a Batteryinverter or Batterysystem is in Island mode, then ems send to this system automatic -100%. The rest must be regulate the function from the batteryinverter. 
//All other battery inverters or battery systems that do not do islanding are treated by the EMS as normal devices with their priorities.
//This EMS can handle 5 device types (Battery, Heating Pump, Electric heating element, Electric charging station and other big consumers)
//This Function receive also Data from a Backend System. In this Backend System runs different ML-Models.
//So its possible that the Backend System controlls the Heating Pumps when its neccessary and also the discharging from the Batterys.
//This make sense when we have bad wheater, less PV-power in the next 24h to switch on the Heating Pumps or cover the consumption.......
//This EMS Function work only with our Backend Communication Library. After 11 Days no communication to our Backend system or no received new HB the Function dissable automatically and set a Message for this at the output
//When we receiven no HB, no Backend Service Ready Flag or an Error from the Backend Service then the Controlling over the Backend is dissabled and the EMS Function run in his "normal" Mode.

//NOTE for diNr.....Designation => 
//_IN = Here Data come in from other Functions or go out to other functions about the GVL
//_OUT = Here Data go out to other functions about the GVL


// V1.1: Added Zero power regulation. Used for CS do use full battery power and then Grid Power
// V1.2: 	Added Operation Mode 4: Adaptive Self Consumption: According to the Battery SOC the operation mode gets switched between self consumtion (EMS mode 1; SOC above setpoint) and load management (EMS mode 3; SOC belwo setpoint) 
//			Operaiton handled via Inpout eOperationMode_Ext 
// 			Added option for disable charging the battery (e.g. for only charging in the night) (b_EnableBatteryChargingControl, b_EnableBatteryChargingControl,b_StartReleaseBatteryCharging,b_StopReleaseBatteryCharging)
// 			Added rMaxBattChargingPower for limiting the maximum battery charge power in percent
//			Made rPeakDetectionforCalculation as input, default 3. This allows different reaction speed of the regulation 
(*------------------------------------------------------------Limits----------------------------------------------------------------------------------*)

stSetupEMS.rSizeMainFuseCS := LIMIT(0,stSetupEMS.rSizeMainFuseCS,500);
stSetupEMS.uiUpdateTime := LIMIT(1,stSetupEMS.uiUpdateTime,600);
stSetupEMS.byResChrgfromGridToBatt := LIMIT(0,stSetupEMS.byResChrgfromGridToBatt,100);
diNrOfEM_IN_ECS := LIMIT(0,diNrOfEM_IN_ECS,Constants_Energy.diMaxNumberOfElectricMeters);
rHeartbeat := LIMIT(0,rHeartbeat,1);
rErrorWarning := LIMIT(0,rErrorWarning,2);
rEnergyOptReady := LIMIT(0,rEnergyOptReady,1);
rNewBattPower := LIMIT(0,rNewBattPower,100000);				
rMaxBattChargingPower := LIMIT(0,rMaxBattChargingPower,100);
rPeakDetectionforCalculation := LIMIT(3,rPeakDetectionforCalculation,100); 

stSetupEMS.rSizeMainFuseCS := DINT_TO_REAL(REAL_TO_DINT(stSetupEMS.rSizeMainFuseCS * 10)) / 10;
		
IF stSetupEMS.byMaxDepthOfDischrgEPO > stSetupEMS.byReserveSOCEPO THEN stSetupEMS.byReserveSOCEPO := stSetupEMS.byMaxDepthOfDischrgEPO + 1; END_IF
IF stSetupEMS.byMaxDepthOfDischrgEPO > stSetupEMS.byPrioMinChrgBattSOCInEPO THEN stSetupEMS.byPrioMinChrgBattSOCInEPO := stSetupEMS.byMaxDepthOfDischrgEPO + 1; END_IF
IF stSetupEMS.byReserveSOCEPO > stSetupEMS.byPrioMinChrgBattSOCInEPO THEN stSetupEMS.byPrioMinChrgBattSOCInEPO := stSetupEMS.byReserveSOCEPO + 1; END_IF
		
stSetupEMS.byMaxDepthOfDischrgEPO := LIMIT(0,stSetupEMS.byMaxDepthOfDischrgEPO,100);
stSetupEMS.byReserveSOCEPO := LIMIT(0,stSetupEMS.byReserveSOCEPO,100);
stSetupEMS.byPrioMinChrgBattSOCInEPO := LIMIT(20,stSetupEMS.byPrioMinChrgBattSOCInEPO,75);


// operation mode handling
IF eOperationMode_Ext = E_OperatingMode_EMS.eAllOff OR eOperationMode_Ext = E_OperatingMode_EMS.eLoadManagement OR eOperationMode_Ext = E_OperatingMode_EMS.ePeakLoadCapping OR eOperationMode_Ext = E_OperatingMode_EMS.eSelfConsumption THEN
	eOperationMode :=  eOperationMode_Ext;
ELSIF eOperationMode_Ext = E_OperatingMode_EMS.eAdaptiveLoadControl THEN
	IF diNumberOfActiveBatterys >= 1 THEN 
		IF DWORD_TO_DINT(dwSumSOC) / diNumberOfActiveBatterys  > by_MinSOC_AdaptiveLC AND NOT b_AnyCarConnected THEN
			eOperationMode := E_OperatingMode_EMS.eSelfConsumption;		// Eigenbedarfsoptimierung
		ELSE
			eOperationMode := E_OperatingMode_EMS.eLoadManagement;		// Lastmanagement
		END_IF  
	END_IF

END_IF

(*-------------------------------------------------------------Calcualte the number of EMS---------------------------------------------------------------*)

//Online change
timDelayStart(IN:= udiCounterOnlineChange_CP <> TwinCAT_SystemInfoVarList._AppInfo.OnlineChangeCnt, PT:= T#15S, Q=> , ET=> );

fbNumberDevice(
	diActualNumberOfDevices:= Lynus_Standards.GVL_Energy.stNumberOfDevices.diNumberOfEMS, 
	diMaxNumberOfDevices:= Constants_Energy.diMaxNumberOfEMS, 
	udiCounterOnlineChange:= TwinCAT_SystemInfoVarList._AppInfo.OnlineChangeCnt, 
	bNumberIsCalculatet=> , 
	bFPNumberIsCalculatet=> , 
	bOnlineChange=> , 
	diNumberForThisDevice=> diNrOfEMS_OUT, 
	diNumberOfTotalDevices=> );

//Write new Numer on GVL
IF fbNumberDevice.bFPNumberIsCalculatet THEN
	Lynus_Standards.GVL_Energy.stNumberOfDevices.diNumberOfEMS := fbNumberDevice.diNumberOfTotalDevices;	
END_IF 

//Delete old Number on GVL
IF fbNumberDevice.bOnlineChange THEN 
	Lynus_Standards.GVL_Energy.stNumberOfDevices.diNumberOfEMS := diNrOfEMS_OUT;	
	udiCounterOnlineChange_CP := TwinCAT_SystemInfoVarList._AppInfo.OnlineChangeCnt; 
END_IF

(*-------------------------------------------------------------Service from Backend is ready and check the connection to backen for dissabel/enable EMS Function---------------------------------------------------------------*)

//Try to reset the variable for connection on the GVL. When all is normal then the Lynus Mqtt connection function set this variable to true in the next cycle
//When we have no connection to the backend or no HB from the Service then after Lynus_Standards.Constants_General.tTimeDissableLynusFunctions days the EMS is dissabled with all of his functionalities
timResetConnectionOnGVL(IN:= NOT timResetConnectionOnGVL.Q, PT:= T#1H, Q=> , ET=> );
IF timResetConnectionOnGVL.Q THEN 
	Lynus_Standards.GVL_Communicator.bStateConnectionToEnableFunctions := FALSE; 
END_IF
IF NOT Lynus_Standards.GVL_Communicator.bStateConnectionToEnableFunctions OR rHeartbeat_CP = rHeartbeat THEN 
	timDissableFunctions.IN := TRUE; 
ELSE 
	timDissableFunctions.IN := FALSE; 
END_IF  
timDissableFunctions(IN:= , PT:= Lynus_Standards.Constants_General.tTimeDissableLynusFunctions, Q=> , ET=> );
	
//Heartbeat, Service Ready and ErrorWarning from Service
timHB(IN:= , PT:= T#130S, Q=> , ET=> );	
IF rHeartbeat <> rHeartbeat_CP THEN 
	timHB.IN := FALSE; 
	rHeartbeat_CP := rHeartbeat; 
ELSE 
	timHB.IN := TRUE; 
END_IF

//Error/Warning Timer and Service Ready Timer
timErrorWarning(IN:= rErrorWarning = 0, PT:= T#10S, Q=> , ET=> );
timEnergyOptReady(IN:= rEnergyOptReady <> 0, PT:= T#10S, Q=> , ET=> );
timControlingState(IN:= bControllingState, PT:= T#10S, Q=> , ET=> );
	
IF timErrorWarning.Q AND timEnergyOptReady.Q AND NOT bControllingState AND NOT timHB.Q AND NOT timDissableFunctions.Q THEN 
	bDischrgCmdFromBackendOK := TRUE; 
END_IF
IF rErrorWarning <> 0 OR rEnergyOptReady = 0 OR timControlingState.Q OR timHB.Q OR timDissableFunctions.Q OR NOT bEnable OR eOperationMode = E_OperatingMode_EMS.eAllOff THEN 
	bDischrgCmdFromBackendOK := FALSE; 
END_IF
	
(*-------------------------------------------------------------Check the number of the device types what are neccessary for EMS---------------------------------------------------------------*)	
	
//To much Devices, Lynus_Standards.Constants_General.tTimeDissableLynusFunctions Days no connection to the backend or Error on the Grid Messurement stop the EMS and set al target power to 0
IF 	Lynus_Standards.GVL_Energy.stNumberOfDevices.diNumberOfEMS > Constants_Energy.diMaxNumberOfEMS OR Lynus_Standards.GVL_Energy.stNumberOfDevices.diNumberOfBatteryInverters > Constants_Energy.diMaxNumberOfBatteryInverters OR
	Lynus_Standards.GVL_Energy.stNumberOfDevices.diNumberOfBatterys > Constants_Energy.diMaxNumberOfBatterys OR Lynus_Standards.GVL_Energy.stNumberOfDevices.diNumberOfECS > Constants_Energy.diMaxNumberOfElectricChargingStations OR
	Lynus_Standards.GVL_Energy.stNumberOfDevices.diNumberOfEHE > Constants_Energy.diMaxNumberOfElectricHeatingElements OR Lynus_Standards.GVL_Energy.stNumberOfDevices.diNumberOfElectricMeters > Constants_Energy.diMaxNumberOfElectricMeters OR
	Lynus_Standards.GVL_Energy.stNumberOfDevices.diNumberOfGenerators > Constants_Energy.diMaxNumberOfGenerators OR Lynus_Standards.GVL_Energy.stNumberOfDevices.diNumberOfGrids > Constants_Energy.diMaxNumberOfGridConnections OR
	Lynus_Standards.GVL_Energy.stNumberOfDevices.diNumberOfHouseConsumption > Constants_Energy.diMaxNumberOfHouseConsumptions OR Lynus_Standards.GVL_Energy.stNumberOfDevices.diNumberOfHP > Constants_Energy.diMaxNumberOfHeatingPumps OR
	Lynus_Standards.GVL_Energy.stNumberOfDevices.diNumberOfOBC > Constants_Energy.diMaxNumberOfOtherBigConsumers OR Lynus_Standards.GVL_Energy.stNumberOfDevices.diNumberOfPvSystems > Constants_Energy.diMaxNumberOfPvSystems OR
	Lynus_Standards.GVL_Sensors.diNumberOfTemperatureSensors > Constants_Sensors.diMaxNumberOfTemperatureSensors OR timDelayStart.Q OR timDissableFunctions.Q OR timErrorGridMessurement.Q THEN 
		bStopAll := TRUE; 
ELSE 
		bStopAll := FALSE;	
END_IF

(*------------------------------------------------------------------------Enable-------------------------------------------------------------------------------*)		
		
bStateEnable := bEnable;

(*--------------------------------------------------------------Allow charging from grid-----------------------------------------------------------------------*)		
		
bStateAllowChrgFromGrid := stSetupEMS.bAllowChrgFromGrid;

(*--------------------------------------------------------------calcualte battery data-----------------------------------------------------------------------*)		
		
//Calcualte the total SOC if we have more then 1 battery in our system
	
diNumberOfActiveBatterys := 0;
dwSumSOC := 0;
FOR liLPBatteryData := 1 TO Constants_Energy.diMaxNumberOfBatterys BY 1 DO
	IF Lynus_Standards.GVL_Energy.stDataOfBatterys[diNrOfEMS_OUT,liLPBatteryData].bEnabled THEN 
		diNumberOfActiveBatterys := diNumberOfActiveBatterys + 1; 
	END_IF
	dwSumSOC := dwSumSOC + Lynus_Standards.GVL_Energy.stDataOfBatterys[diNrOfEMS_OUT,liLPBatteryData].dwSOC;
END_FOR
	
dwSumSOCInEPO := 0;
FOR liLPSumSOCInEPO := 1 TO Constants_Energy.diMaxNumberOfBatteryInverters BY 1 DO
	IF Lynus_Standards.GVL_Energy.stDataOfBatteryInverters[diNrOfEMS_OUT,liLPSumSOCInEPO].bWorkOnIslandMode THEN 
		dwSumSOCInEPO := dwSumSOCInEPO + Lynus_Standards.GVL_Energy.stDataOfBatteryInverters[diNrOfEMS_OUT,liLPSumSOCInEPO].dwBatterySOC; 
	END_IF
END_FOR		
		
IF diNumberOfActiveBatterys > 0 THEN
	dwAvarageBatterySOC := DINT_TO_DWORD(DWORD_TO_DINT(dwSumSOC) / diNumberOfActiveBatterys);
END_IF

//Check if one or more Batterysystems or batteryinverter make island mode

diNumberOfBatteryInverterInEPO := 0;
FOR liLPInEPO := 1 TO Constants_Energy.diMaxNumberOfBatteryInverters BY 1 DO
	IF Lynus_Standards.GVL_Energy.stDataOfBatteryInverters[diNrOfEMS_OUT,liLPInEPO].bWorkOnIslandMode THEN 
		bEPMActive := TRUE; diNumberOfBatteryInverterInEPO := diNumberOfBatteryInverterInEPO + 1; 
	END_IF
END_FOR 

IF diNumberOfBatteryInverterInEPO > 0 THEN
	dwAvarageBatterySOCInEPO := DINT_TO_DWORD(DWORD_TO_DINT(dwSumSOCInEPO) / diNumberOfBatteryInverterInEPO);
ELSE
	dwAvarageBatterySOCInEPO := 0;
END_IF
	
IF diNumberOfBatteryInverterInEPO <= 0 THEN bEPMActive := FALSE; END_IF

//Check the max. power of the grid connection and the sum of grid power
lrSizeGridConnection := 0;
lrGridPower := 0;
bErrorOnGridMessurement := FALSE;
FOR liLPGridData := 1 TO Constants_Energy.diMaxNumberOfGridConnections BY 1 DO
	lrSizeGridConnection := lrSizeGridConnection + Lynus_Standards.GVL_Energy.stDataGridConnections[diNrOfEMS_OUT,liLPGridData].rSizeGridConn;
	lrGridPower := lrGridPower + Lynus_Standards.GVL_Energy.stDataGridConnections[diNrOfEMS_OUT,liLPGridData].lrPower;
	IF Lynus_Standards.GVL_Energy.stDataGridConnections[diNrOfEMS_OUT,liLPGridData].byErrorWarning = 2 THEN 
		bErrorOnGridMessurement := TRUE; 
	END_IF 
END_FOR

//Error on Grid Messurement. (Stop the EMS Function)
timErrorGridMessurement(IN:= bErrorOnGridMessurement, PT:= T#30S, Q=> , ET=> );
	
//Timer for peaks to cut this
timCutPeaks(IN:= , PT:= T#2.5S, Q=> , ET=> );	

(*--------------------------------------------------------------Timeout-----------------------------------------------------------------------*)	

//Timout is using to go on next step if somthing goes wrong in the steps in what we check the next priority from the several devices
IF uiState = uiState_CP AND uiState >= 30 AND uiState <= 110 THEN 
	timTimeout.IN := TRUE; 
ELSE 
	timTimeout.IN := FALSE; 
END_IF
//Choose the right Delay. Depending from the maximum of allowed Devices
diBiggestNumberOfDeviceConstants := 0;
IF Constants_Energy.diMaxNumberOfBatterys > diBiggestNumberOfDeviceConstants THEN 
	diBiggestNumberOfDeviceConstants := Constants_Energy.diMaxNumberOfBatterys; 
END_IF
IF Constants_Energy.diMaxNumberOfBatteryInverters > diBiggestNumberOfDeviceConstants THEN 
	diBiggestNumberOfDeviceConstants := Constants_Energy.diMaxNumberOfBatteryInverters; 
END_IF 
IF Constants_Energy.diMaxNumberOfElectricHeatingElements > diBiggestNumberOfDeviceConstants THEN 
	diBiggestNumberOfDeviceConstants := Constants_Energy.diMaxNumberOfElectricHeatingElements; 
END_IF
IF Constants_Energy.diMaxNumberOfHeatingPumps > diBiggestNumberOfDeviceConstants THEN 
	diBiggestNumberOfDeviceConstants := Constants_Energy.diMaxNumberOfHeatingPumps; 
END_IF
IF Constants_Energy.diMaxNumberOfElectricChargingStations > diBiggestNumberOfDeviceConstants THEN 
	diBiggestNumberOfDeviceConstants := Constants_Energy.diMaxNumberOfElectricChargingStations; 
END_IF
IF Constants_Energy.diMaxNumberOfOtherBigConsumers > diBiggestNumberOfDeviceConstants THEN 
	diBiggestNumberOfDeviceConstants := Constants_Energy.diMaxNumberOfOtherBigConsumers; 
END_IF 

//Cycletime in MS
fbTaskIndex(index=> );
udiCycleTime := TwinCAT_SystemInfoVarList._TaskInfo[fbTaskIndex.index].CycleTime / 10000;
//Make a caculation with max Prio Number of 255, the cycle time and the biggest number. Because in the dumbest case it can take so long in one step until all priorities are gone through.
timTimeout.PT := (T#1MS * udiCycleTime * 255 * diBiggestNumberOfDeviceConstants) + T#10S; 
timTimeout(IN:= , PT:= , Q=> , ET=> );

(*--------------------------------------------------------------Timer for Battery-----------------------------------------------------------------------*)

//This timer ensures that the respective battery is full and thus in case of surplus or no surplus the power setting is directly regulated to 0% or -99.99% to accelerate the process.
//See in Step 131
//Only important in the self consumption mode

FOR liLPDataBatteryInverter := 1 TO Constants_Energy.diMaxNumberOfBatteryInverters BY 1 DO
	IF Lynus_Standards.GVL_Energy.stDataOfBatteryInverters[diNrOfEMS_OUT,liLPDataBatteryInverter].dwBatterySOC >= 100 THEN
		arrTimBatterysAreFull[liLPDataBatteryInverter](IN:= TRUE, PT:= T#2M, Q=> , ET=> );
	ELSE
		arrTimBatterysAreFull[liLPDataBatteryInverter](IN:= FALSE, PT:= T#2M, Q=> , ET=> );
	END_IF						
END_FOR
	
(*-------------------------------------------------------------Logic form the ems function to manage the devices-----------------------------------------------------------------------------------*)		
		
timCalculateNewPowerValue(IN:= bEnable AND NOT timCalculateNewPowerValue.Q AND uiState = 10, PT:= (T#1S * stSetupEMS.uiUpdateTime) , Q=> , ET=> );		

IF NOT bEnable OR FPEPO.Q OR FNEPO.Q OR diMemCmpOperationState <> 0 OR eOperationMode = E_OperatingMode_EMS.eAllOff OR bStopAll THEN 
	uiState := 0; 
END_IF
IF stSetupEMS.rSizeMainFuseCS <> rSizeMainFuseCS_CP OR diNrOfEM_IN_ECS <> diNrOfEM_IN_CS_CP THEN 
	uiState := 1; 
END_IF

CASE uiState OF
	
	0: //Init Step
		
		byProgress := 0;
	
		eOperationModeEMS_CP := eOperationMode;
	
		IF bEnable AND eOperationMode <> E_OperatingMode_EMS.eAllOff AND NOT bStopAll THEN 
			uiState := 10; 
			arrActualPrioInTurn[1] := 1; arrActualPrioInTurn[2] := 1; arrActualPrioInTurn[3] := 1; arrActualPrioInTurn[4] := 1; arrActualPrioInTurn[5] := 1;
			arrActualStepInTurn[1] := 1; arrActualStepInTurn[2] := 1; 
			arrActualStepInTurn_CP[1]:= arrActualStepInTurn[1];
			arrActualStepInTurn_CP[2] := arrActualStepInTurn[2];
			bySmGrActiveCommonPrio_CP := 1;	liCounterCkeckDeviceAndPrio := 0;
			arrCTCheckActivePrio[1] := 0; arrCTCheckActivePrio[2] := 0; arrCTCheckActivePrio[3] := 0; arrCTCheckActivePrio[4] := 0; arrCTCheckActivePrio[5] := 0; liNrOfNotDoneDevices := 0; diNumberOfDevicesFromEachType := 0;
			timCutPeaks.IN := FALSE;
			arrMinPrioReached[1] := TRUE; arrMinPrioReached[2] := TRUE; arrMinPrioReached[3] := TRUE; arrMinPrioReached[4] := TRUE; arrMinPrioReached[5] := TRUE;
			arrMaxPrioReached[1] := FALSE; arrMaxPrioReached[2] := FALSE; arrMaxPrioReached[3] := FALSE; arrMaxPrioReached[4] := FALSE; arrMaxPrioReached[5] := FALSE;
		END_IF
		
	1: 	//Set the battery to Init if some Inputs are missing between the operation	
		arrActualPrioInTurn[1] := 1;
		bySmGrActiveCommonPrio_CP := 1;	
		arrCTCheckActivePrio[1] := 0; arrCTCheckActivePrio[2] := 0; arrCTCheckActivePrio[3] := 0; arrCTCheckActivePrio[4] := 0; arrCTCheckActivePrio[5] := 0; liNrOfNotDoneDevices := 0; diNumberOfDevicesFromEachType := 0; liCounterCkeckDeviceAndPrio := 0;
		timCutPeaks.IN := FALSE;
		arrMinPrioReached[1] := TRUE;
		arrMaxPrioReached[1] := FALSE;
		rSizeMainFuseCS_CP := stSetupEMS.rSizeMainFuseCS;
		diNrOfEM_IN_CS_CP := diNrOfEM_IN_ECS;
		uiState := 10;

	10: //After the timer is expired then ckeck if we have surplus or not
		//Surplus calculation in the Self consumption mode 
		IF NOT bEPMActive AND eOperationMode = E_OperatingMode_EMS.eSelfConsumption THEN	
			lrActualSurplusOrConsumption := 0;
			FOR liLPActualSurplusOrConsumption := 1 TO Constants_Energy.diMaxNumberOfGridConnections BY 1 DO
				lrActualSurplusOrConsumption := lrActualSurplusOrConsumption + Lynus_Standards.GVL_Energy.stDataGridConnections[diNrOfEMS_OUT,liLPActualSurplusOrConsumption].lrPower;
			END_FOR
			IF lrActualSurplusOrConsumption < - Constants_Energy.rToleranceSurplusConsumption THEN 
				bSurplusAvailable := TRUE; 
			END_IF
			IF lrActualSurplusOrConsumption >= Constants_Energy.rToleranceSurplusConsumption THEN 
				bSurplusAvailable := FALSE; 
			END_IF
			IF lrActualSurplusOrConsumption >= - Constants_Energy.rToleranceSurplusConsumption AND lrActualSurplusOrConsumption < Constants_Energy.rToleranceSurplusConsumption THEN 
				bSurplusAvailable := FALSE; lrActualSurplusOrConsumption := 0; 
			END_IF
				
			//Peaks from <> 3 KW activate timer to wait 2.5 seconds before calculate
			IF lrActualSurplusOrConsumption >= (lrActualSurplusOrConsumptionOld + 3) OR lrActualSurplusOrConsumption <= (lrActualSurplusOrConsumptionOld - 3) THEN 
				timCutPeaks.IN := TRUE; 
			ELSE 
				timCutPeaks.IN := FALSE; 
			END_IF 
			lrActualSurplusOrConsumptionOld := lrActualSurplusOrConsumption;	
				
			IF timCalculateNewPowerValue.Q AND NOT timCutPeaks.Q AND rControllerQPIDSC <= 0 AND NOT fbPIDDischrgCmdFromBackend.bEnable THEN 
				uiState := 30; 
			END_IF
		END_IF
		
		//Surplus calculation in the peak load capping mode 
		IF NOT bEPMActive AND eOperationMode = E_OperatingMode_EMS.ePeakLoadCapping THEN	
			lrActualSurplusOrConsumption := 0;
			FOR liLPActualSurplusOrConsumption := 1 TO Constants_Energy.diMaxNumberOfGridConnections BY 1 DO
				lrActualSurplusOrConsumption := lrActualSurplusOrConsumption + Lynus_Standards.GVL_Energy.stDataGridConnections[diNrOfEMS_OUT,liLPActualSurplusOrConsumption].lrPower;
			END_FOR
			
			lrActualSurplusOrConsumption := (lrSizeGridConnection) - lrActualSurplusOrConsumption;
			lrActualSurplusOrConsumption := lrActualSurplusOrConsumption * - 1;
			
			IF lrActualSurplusOrConsumption < - Constants_Energy.rToleranceSurplusConsumption THEN 
				bSurplusAvailable := TRUE; 
			END_IF
			IF lrActualSurplusOrConsumption >= Constants_Energy.rToleranceSurplusConsumption THEN 
				bSurplusAvailable := FALSE; 
			END_IF	
			IF lrActualSurplusOrConsumption >= - Constants_Energy.rToleranceSurplusConsumption AND lrActualSurplusOrConsumption < Constants_Energy.rToleranceSurplusConsumption THEN 
				bSurplusAvailable := FALSE; lrActualSurplusOrConsumption := 0; 
			END_IF
		
			//Peaks from <> 3 KW activate timer to wait 2.5 seconds before calculate
			IF lrActualSurplusOrConsumption >= (lrActualSurplusOrConsumptionOld + 3) OR lrActualSurplusOrConsumption <= (lrActualSurplusOrConsumptionOld - 3) THEN 
				timCutPeaks.IN := TRUE; 
			ELSE 
				timCutPeaks.IN := FALSE; 
			END_IF 
			lrActualSurplusOrConsumptionOld := lrActualSurplusOrConsumption;
		
			IF timCalculateNewPowerValue.Q AND NOT timCutPeaks.Q THEN 
				uiState := 50; 
				//Set here to 0 because if other devices has Prio 1 or 255 the EMS not can finsih the Step why we leave Step 30
				liNrOfNotDoneDevices := 0; 
				//On this Operation Mode the batterys are always active. So we dont need the Step 30. See the PID Controllers for this mode
				IF ((bSurplusAvailable AND diNumberOfDevicesFromEachType = 0) OR (diNumberOfActiveBatterys = 0 AND bSurplusAvailable) OR (diNumberOfActiveBatterys <> 0 AND bSurplusAvailable)) THEN 
					arrActualPrioInTurn[1] := 255; 
					arrMinPrioReached[1] := FALSE; 
					arrMaxPrioReached[1] := TRUE; 
				END_IF
				IF ((NOT bSurplusAvailable AND diNumberOfDevicesFromEachType = 0) OR (diNumberOfActiveBatterys = 0 AND NOT bSurplusAvailable) OR (diNumberOfActiveBatterys <> 0 AND NOT bSurplusAvailable)) THEN 
					arrActualPrioInTurn[1] := 1; 
					arrMinPrioReached[1] := TRUE; 
					arrMaxPrioReached[1] := FALSE; 
				END_IF
			END_IF;
		END_IF
		
		//Surplus calculation in the load managemant mode 
		IF NOT bEPMActive AND eOperationMode = E_OperatingMode_EMS.eLoadManagement THEN	
			lrActualSurplusOrConsumption := 0;
			FOR liLPActualSurplusOrConsumption := 1 TO Constants_Energy.diMaxNumberOfGridConnections BY 1 DO
				lrActualSurplusOrConsumption := lrActualSurplusOrConsumption + Lynus_Standards.GVL_Energy.stDataGridConnections[diNrOfEMS_OUT,liLPActualSurplusOrConsumption].lrPower;
			END_FOR
				
			lrActualSurplusOrConsumption := (lrSizeGridConnection) - lrActualSurplusOrConsumption;
			lrActualSurplusOrConsumption := lrActualSurplusOrConsumption * - 1;
			
			IF lrActualSurplusOrConsumption < - Constants_Energy.rToleranceSurplusConsumption THEN 
				bSurplusAvailable := TRUE; 
			END_IF
			IF lrActualSurplusOrConsumption >= Constants_Energy.rToleranceSurplusConsumption THEN 
				bSurplusAvailable := FALSE; 
			END_IF	
			IF lrActualSurplusOrConsumption >= - Constants_Energy.rToleranceSurplusConsumption AND lrActualSurplusOrConsumption < Constants_Energy.rToleranceSurplusConsumption THEN 
				bSurplusAvailable := FALSE; lrActualSurplusOrConsumption := 0; 
			END_IF
			
			//Peaks from <> 3 KW activate timer to wait 2.5 seconds before calculate
			IF lrActualSurplusOrConsumption >= (lrActualSurplusOrConsumptionOld + 3) OR lrActualSurplusOrConsumption <= (lrActualSurplusOrConsumptionOld - 3) THEN 
				timCutPeaks.IN := TRUE; 
			ELSE 
				timCutPeaks.IN := FALSE; 
			END_IF 
			lrActualSurplusOrConsumptionOld := lrActualSurplusOrConsumption;
			
			IF timCalculateNewPowerValue.Q AND NOT timCutPeaks.Q THEN 
				uiState := 50; 
				//Set here to 0 because if other devices has Prio 1 or 255 the EMS not can finsih the Step why we leave Step 30
				liNrOfNotDoneDevices := 0; 
				//On this Operation Mode the batterys are always active. So we dont need the Step 30. See the PID Controllers for this mode
				IF ((bSurplusAvailable AND diNumberOfDevicesFromEachType = 0) OR (diNumberOfActiveBatterys = 0 AND bSurplusAvailable) OR (diNumberOfActiveBatterys <> 0 AND bSurplusAvailable)) THEN 
					arrActualPrioInTurn[1] := 255; 
					arrMinPrioReached[1] := FALSE; 
					arrMaxPrioReached[1] := TRUE; 
				END_IF
				IF ((NOT bSurplusAvailable AND diNumberOfDevicesFromEachType = 0) OR (diNumberOfActiveBatterys = 0 AND NOT bSurplusAvailable) OR (diNumberOfActiveBatterys <> 0 AND NOT bSurplusAvailable)) THEN 
					arrActualPrioInTurn[1] := 1; 
					arrMinPrioReached[1] := TRUE; 
					arrMaxPrioReached[1] := FALSE; 
				END_IF
			END_IF
		END_IF
		
		//Surplus calculation in the emergency power mode
		IF bEPMActive THEN	
			lrActualSurplusOrConsumption := 0;
			FOR liLPActualSurplusOrConsumption := 1 TO Constants_Energy.diMaxNumberOfBatteryInverters BY 1 DO
				IF Lynus_Standards.GVL_Energy.stDataOfBatteryInverters[diNrOfEMS_OUT,liLPActualSurplusOrConsumption].bWorkOnIslandMode THEN lrActualSurplusOrConsumption := lrActualSurplusOrConsumption + Lynus_Standards.GVL_Energy.stDataOfBatteryInverters[diNrOfEMS_OUT,liLPActualSurplusOrConsumption].lrPowerOnIslandMode; END_IF
			END_FOR
			IF lrActualSurplusOrConsumption < - Constants_Energy.rToleranceSurplusConsumption THEN 
				bSurplusAvailable := TRUE; 
			END_IF
			IF lrActualSurplusOrConsumption >= Constants_Energy.rToleranceSurplusConsumption THEN 
				bSurplusAvailable := FALSE; 
			END_IF
			IF lrActualSurplusOrConsumption >= - Constants_Energy.rToleranceSurplusConsumption AND lrActualSurplusOrConsumption < Constants_Energy.rToleranceSurplusConsumption THEN 
				bSurplusAvailable := FALSE; 
				lrActualSurplusOrConsumption := 0; 
			END_IF
			
			//Peaks from <> 3 KW activate timer to wait 2.5 seconds before calculate
			IF lrActualSurplusOrConsumption >= (lrActualSurplusOrConsumptionOld + 3) OR lrActualSurplusOrConsumption <= (lrActualSurplusOrConsumptionOld - 3) THEN 
				timCutPeaks.IN := TRUE; 
			ELSE 
				timCutPeaks.IN := FALSE; 
			END_IF 
			lrActualSurplusOrConsumptionOld := lrActualSurplusOrConsumption;
			
			IF timCalculateNewPowerValue.Q AND NOT timCutPeaks.Q AND rControllerQPIDEPO <= 0 THEN 
				uiState := 21; 
			END_IF;
		END_IF
		
	21:	//If emergency power is active then first charge batteries that are build the island mode until byPrioMinChargeBattSOCInEPO, only then start normal mode according to priorities. 
		//Batterys or battery inverters that do not work on island mode, are only loaded afterwards based on the priority.  
		//As long as this SOC from byPrioMinChargeBattSOCInEPO is undercut, all other devices are regulated to 0.
		IF dwAvarageBatterySOCInEPO < stSetupEMS.byPrioMinChrgBattSOCInEPO THEN
			uiState := 0;
			bSurplusAvailable := FALSE;
			lrActualSurplusOrConsumption := 0;
			arrMinPrioReached[1] := TRUE; 
			arrMinPrioReached[2] := TRUE; 
			arrMinPrioReached[3] := TRUE; 
			arrMinPrioReached[4] := TRUE; 
			arrMinPrioReached[5] := TRUE;
			arrMaxPrioReached[1] := FALSE; 
			arrMaxPrioReached[2] := FALSE; 
			arrMaxPrioReached[3] := FALSE; 
			arrMaxPrioReached[4] := FALSE; 
			arrMaxPrioReached[5] := FALSE;
			bChargePrioBatterysOnEPO := TRUE;
		END_IF
		IF 	(dwAvarageBatterySOCInEPO >= (stSetupEMS.byPrioMinChrgBattSOCInEPO + 1) AND stSetupEMS.byPrioMinChrgBattSOCInEPO < 75) OR
			(dwAvarageBatterySOCInEPO >= stSetupEMS.byPrioMinChrgBattSOCInEPO AND stSetupEMS.byPrioMinChrgBattSOCInEPO >= 75) THEN
				bChargePrioBatterysOnEPO := FALSE;
				uiState := 30;
		END_IF
		
	30: //Check the priority for battery or battery inverters to controll (Batterys they are in island mode are not considered here)
		uiState_CP := uiState;
		
		//First check if we have min 1 of this Device Type. If not, complete this Device Type and go to the next step
		//Check also the bigest Priority of this Device Type
		diNumberOfDevicesFromEachType := 0; bySearchBigestPrio := 0;
		FOR liLPCheckDeviceAndPrio := 1 TO Constants_Energy.diMaxNumberOfBatteryInverters BY 1 DO
			IF Lynus_Standards.GVL_Energy.stDataOfBatteryInverters[diNrOfEMS_OUT,liLPCheckDeviceAndPrio].byPriority <> 0 THEN 
				diNumberOfDevicesFromEachType := diNumberOfDevicesFromEachType + 1; 
			END_IF
			IF Lynus_Standards.GVL_Energy.stDataOfBatteryInverters[diNrOfEMS_OUT,liLPCheckDeviceAndPrio].byPriority > bySearchBigestPrio THEN 
				bySearchBigestPrio := Lynus_Standards.GVL_Energy.stDataOfBatteryInverters[diNrOfEMS_OUT,liLPCheckDeviceAndPrio].byPriority; 
			END_IF  	
		END_FOR 
		IF bSurplusAvailable AND arrActualPrioInTurn[1] > bySearchBigestPrio AND uiState = 30 THEN 
			arrActualPrioInTurn[1] := 255; 
		END_IF
		IF NOT bSurplusAvailable AND arrActualPrioInTurn[1] > bySearchBigestPrio AND uiState = 30 THEN 
			arrActualPrioInTurn[1] := bySearchBigestPrio; 
		END_IF     
		
		IF bSurplusAvailable AND diNumberOfDevicesFromEachType = 0 THEN 
			arrActualPrioInTurn[1] := 255; 
		END_IF
		IF NOT bSurplusAvailable AND diNumberOfDevicesFromEachType = 0 THEN 
			arrActualPrioInTurn[1] := 1; 
		END_IF
		
		//Count up each Device
		arrCTCheckActivePrio[1] := arrCTCheckActivePrio[1] + 1;
		arrCTCheckActivePrio[1] := LIMIT(1,arrCTCheckActivePrio[1],Constants_Energy.diMaxNumberOfBatteryInverters);		
				
		//Surplus
		IF bSurplusAvailable AND Lynus_Standards.GVL_Energy.stDataOfBatteryInverters[diNrOfEMS_OUT,arrCTCheckActivePrio[1]].byPriority = arrActualPrioInTurn[1] AND Lynus_Standards.GVL_Energy.stDataOfBatteryInverters[diNrOfEMS_OUT,arrCTCheckActivePrio[1]].rTargetPowerEMS > -100 AND NOT Lynus_Standards.GVL_Energy.stDataOfBatteryInverters[diNrOfEMS_OUT,arrCTCheckActivePrio[1]].bWorkOnIslandMode THEN
			arrMaxPrioReached[1] := FALSE;
			arrMinPrioReached[1] := FALSE;
			arrCTCheckActivePrio[1] := 0; 
			liNrOfNotDoneDevices := 0; 
			liCounterCkeckDeviceAndPrio := 0; //Set here to 0 because in next Step we dont can work with a loop (performance Problems on small PLC)
			uiState := 50;
		ELSE
			IF bSurplusAvailable AND arrActualPrioInTurn[1] < 255 AND uiState = 30 AND arrCTCheckActivePrio[1] = Constants_Energy.diMaxNumberOfBatteryInverters THEN 
				arrActualPrioInTurn[1] := arrActualPrioInTurn[1] + 1; 
				arrCTCheckActivePrio[1] := 0; 
			END_IF
		END_IF
			//No surplus
		IF NOT bSurplusAvailable AND Lynus_Standards.GVL_Energy.stDataOfBatteryInverters[diNrOfEMS_OUT,arrCTCheckActivePrio[1]].byPriority = arrActualPrioInTurn[1] AND Lynus_Standards.GVL_Energy.stDataOfBatteryInverters[diNrOfEMS_OUT,arrCTCheckActivePrio[1]].rTargetPowerEMS < 0 AND NOT Lynus_Standards.GVL_Energy.stDataOfBatteryInverters[diNrOfEMS_OUT,arrCTCheckActivePrio[1]].bWorkOnIslandMode THEN
			arrMaxPrioReached[1] := FALSE;
			arrMinPrioReached[1] := FALSE;
			arrCTCheckActivePrio[1] := 0; 
			liNrOfNotDoneDevices := 0; 
			liCounterCkeckDeviceAndPrio := 0;
			uiState := 50;
		ELSE
			IF NOT bSurplusAvailable AND arrActualPrioInTurn[1] > 1 AND uiState = 30 AND arrCTCheckActivePrio[1] = Constants_Energy.diMaxNumberOfBatteryInverters THEN 
				arrActualPrioInTurn[1] := arrActualPrioInTurn[1] - 1; 
				arrCTCheckActivePrio[1] := 0; 
			END_IF
		END_IF

	//Go to next step if we are on min prio or on max prio and the target power is just set to the min or to the max value.
		liNrOfNotDoneDevices := 0;
		IF uiState = 30 THEN
			FOR liLPCheckDeviceAndPrio := 1 TO Constants_Energy.diMaxNumberOfBatteryInverters BY 1 DO
				IF arrActualPrioInTurn[1] = 1 AND Lynus_Standards.GVL_Energy.stDataOfBatteryInverters[diNrOfEMS_OUT,liLPCheckDeviceAndPrio].rTargetPowerEMS <> 0 AND Lynus_Standards.GVL_Energy.stDataOfBatteryInverters[diNrOfEMS_OUT,liLPCheckDeviceAndPrio].byPriority = 1 THEN
					liNrOfNotDoneDevices := liNrOfNotDoneDevices + 1;	
				END_IF
				IF arrActualPrioInTurn[1] = 255 AND Lynus_Standards.GVL_Energy.stDataOfBatteryInverters[diNrOfEMS_OUT,liLPCheckDeviceAndPrio].rTargetPowerEMS > - 100 AND Lynus_Standards.GVL_Energy.stDataOfBatteryInverters[diNrOfEMS_OUT,liLPCheckDeviceAndPrio].byPriority = 255 THEN
					liNrOfNotDoneDevices := liNrOfNotDoneDevices + 1;	
				END_IF
			END_FOR	
		END_IF
	
		IF arrActualPrioInTurn[1] = 1 AND uiState = 30 AND liNrOfNotDoneDevices = 0 AND arrCTCheckActivePrio[1] = Constants_Energy.diMaxNumberOfBatteryInverters THEN 
			arrMinPrioReached[1] := TRUE; 
			arrMaxPrioReached[1] := FALSE; 
			liNrOfNotDoneDevices := 0; 
			uiState := 50; 
			arrCTCheckActivePrio[1] := 0; 
			liCounterCkeckDeviceAndPrio := 0;
		END_IF
		IF arrActualPrioInTurn[1] = 255 AND uiState = 30 AND liNrOfNotDoneDevices = 0 AND arrCTCheckActivePrio[1] = Constants_Energy.diMaxNumberOfBatteryInverters THEN 
			arrMaxPrioReached[1] := TRUE; 
			arrMinPrioReached[1] := FALSE; 
			liNrOfNotDoneDevices := 0; 
			uiState := 50; 
			arrCTCheckActivePrio[1] := 0; 
			liCounterCkeckDeviceAndPrio := 0;
		END_IF
		
		//Timout, go to next step
		IF timTimeout.Q AND uiState = 30 THEN 
			uiState := 50; 
		END_IF
		
	50: //Check the priority for the heating pump incl. the steps to controll it
		uiState_CP := uiState;	
	
		//Counter to ckeck if we reached at the min or the max prio
		IF uiState = 50 THEN 
			liCounterCkeckDeviceAndPrio := liCounterCkeckDeviceAndPrio + 1; 
		END_IF
	
		//First check if we have min 1 of this Device Type. If not, complete this Device Type and go to the next step
		//Check also the bigest Priority of this Device Type
		diNumberOfDevicesFromEachType := 0; bySearchBigestPrio := 0;
		FOR liLPCheckDeviceAndPrio := 1 TO Constants_Energy.diMaxNumberOfHeatingPumps BY 1 DO
			IF Lynus_Standards.GVL_Energy.stDataHeatingPumps[diNrOfEMS_OUT,liLPCheckDeviceAndPrio].byPriority <> 0 THEN 
				diNumberOfDevicesFromEachType := diNumberOfDevicesFromEachType + 1; 
			END_IF
			IF Lynus_Standards.GVL_Energy.stDataHeatingPumps[diNrOfEMS_OUT,liLPCheckDeviceAndPrio].byPriority > bySearchBigestPrio THEN 
				bySearchBigestPrio := Lynus_Standards.GVL_Energy.stDataHeatingPumps[diNrOfEMS_OUT,liLPCheckDeviceAndPrio].byPriority; 
			END_IF  
		END_FOR 
		IF bSurplusAvailable AND arrActualPrioInTurn[2] > bySearchBigestPrio AND uiState = 50 THEN 
			arrActualPrioInTurn[2] := 255; 
		END_IF
		IF NOT bSurplusAvailable AND arrActualPrioInTurn[2] > bySearchBigestPrio AND uiState = 50 THEN 
			arrActualPrioInTurn[2] := bySearchBigestPrio; 
		END_IF
	
		IF bSurplusAvailable AND diNumberOfDevicesFromEachType = 0 THEN 
			arrActualPrioInTurn[2] := 255; 
		END_IF
		IF NOT bSurplusAvailable AND diNumberOfDevicesFromEachType = 0 THEN 
			arrActualPrioInTurn[2] := 1; 
		END_IF
	
		//Count up each Device
		arrCTCheckActivePrio[2] := arrCTCheckActivePrio[2] + 1;
		arrCTCheckActivePrio[2] := LIMIT(1,arrCTCheckActivePrio[2],Constants_Energy.diMaxNumberOfHeatingPumps);
	
		//Surplus
		IF bSurplusAvailable AND Lynus_Standards.GVL_Energy.stDataHeatingPumps[diNrOfEMS_OUT,arrCTCheckActivePrio[2]].byPriority = arrActualPrioInTurn[2] AND NOT Lynus_Standards.GVL_Energy.stDataHeatingPumps[diNrOfEMS_OUT,arrCTCheckActivePrio[2]].bIsStepSwitched AND NOT 
		Lynus_Standards.GVL_Energy.stDataHeatingPumps[diNrOfEMS_OUT,arrCTCheckActivePrio[2]].bIsControllable AND Lynus_Standards.GVL_Energy.stDataHeatingPumps[diNrOfEMS_OUT,arrCTCheckActivePrio[2]].arrTargetPowerEMS[1] < 100 THEN
			arrActualStepInTurn[1] := 1;	
			arrMaxPrioReached[2] := FALSE;
			arrMinPrioReached[2] := FALSE;
			arrCTCheckActivePrio[2] := 0; 
			liNrOfNotDoneDevices := 0; 
			liCounterCkeckDeviceAndPrio := 0; //Set here to 0 because in next Step we dont can work with a loop (performance Problems on small PLC)
			uiState := 70;
		ELSIF bSurplusAvailable AND Lynus_Standards.GVL_Energy.stDataHeatingPumps[diNrOfEMS_OUT,arrCTCheckActivePrio[2]].byPriority = arrActualPrioInTurn[2] AND Lynus_Standards.GVL_Energy.stDataHeatingPumps[diNrOfEMS_OUT,arrCTCheckActivePrio[2]].byNumberOfSteps = 0 AND
		Lynus_Standards.GVL_Energy.stDataHeatingPumps[diNrOfEMS_OUT,arrCTCheckActivePrio[2]].arrTargetPowerEMS[1] < 100 THEN 
			arrActualStepInTurn[1] := 1;	
			arrMaxPrioReached[2] := FALSE;
			arrMinPrioReached[2] := FALSE;
			arrCTCheckActivePrio[2] := 0; 
			liNrOfNotDoneDevices := 0; 
			liCounterCkeckDeviceAndPrio := 0;
			uiState := 70;
		ELSIF bSurplusAvailable AND Lynus_Standards.GVL_Energy.stDataHeatingPumps[diNrOfEMS_OUT,arrCTCheckActivePrio[2]].byPriority = arrActualPrioInTurn[2] AND NOT Lynus_Standards.GVL_Energy.stDataHeatingPumps[diNrOfEMS_OUT,arrCTCheckActivePrio[2]].bIsStepSwitched AND 
		Lynus_Standards.GVL_Energy.stDataHeatingPumps[diNrOfEMS_OUT,arrCTCheckActivePrio[2]].bIsControllable AND Lynus_Standards.GVL_Energy.stDataHeatingPumps[diNrOfEMS_OUT,arrCTCheckActivePrio[2]].arrTargetPowerEMS[1] < 100 THEN 
			arrActualStepInTurn[1] := 1;	
			arrMaxPrioReached[2] := FALSE;
			arrMinPrioReached[2] := FALSE;
			arrCTCheckActivePrio[2] := 0; 
			liNrOfNotDoneDevices := 0; 
			liCounterCkeckDeviceAndPrio := 0;
			uiState := 70;
		ELSIF bSurplusAvailable AND Lynus_Standards.GVL_Energy.stDataHeatingPumps[diNrOfEMS_OUT,arrCTCheckActivePrio[2]].byPriority = arrActualPrioInTurn[2] AND Lynus_Standards.GVL_Energy.stDataHeatingPumps[diNrOfEMS_OUT,arrCTCheckActivePrio[2]].bIsStepSwitched AND 
		Lynus_Standards.GVL_Energy.stDataHeatingPumps[diNrOfEMS_OUT,arrCTCheckActivePrio[2]].bIsControllable AND Lynus_Standards.GVL_Energy.stDataHeatingPumps[diNrOfEMS_OUT,arrCTCheckActivePrio[2]].byNumberOfSteps = 1 AND Lynus_Standards.GVL_Energy.stDataHeatingPumps[diNrOfEMS_OUT,arrCTCheckActivePrio[2]].arrTargetPowerEMS[1] < 100 THEN 
			arrActualStepInTurn[1] := 1;	
			arrMaxPrioReached[2] := FALSE;
			arrMinPrioReached[2] := FALSE;
			arrCTCheckActivePrio[2] := 0; 
			liNrOfNotDoneDevices := 0; 
			liCounterCkeckDeviceAndPrio := 0;
			uiState := 70;
		ELSIF bSurplusAvailable AND Lynus_Standards.GVL_Energy.stDataHeatingPumps[diNrOfEMS_OUT,arrCTCheckActivePrio[2]].byPriority = arrActualPrioInTurn[2] AND Lynus_Standards.GVL_Energy.stDataHeatingPumps[diNrOfEMS_OUT,arrCTCheckActivePrio[2]].bIsStepSwitched AND 
		Lynus_Standards.GVL_Energy.stDataHeatingPumps[diNrOfEMS_OUT,arrCTCheckActivePrio[2]].bIsControllable AND Lynus_Standards.GVL_Energy.stDataHeatingPumps[diNrOfEMS_OUT,arrCTCheckActivePrio[2]].byNumberOfSteps = 2 AND (Lynus_Standards.GVL_Energy.stDataHeatingPumps[diNrOfEMS_OUT,arrCTCheckActivePrio[2]].arrTargetPowerEMS[1] < 100 OR Lynus_Standards.GVL_Energy.stDataHeatingPumps[diNrOfEMS_OUT,arrCTCheckActivePrio[2]].arrTargetPowerEMS[2] < 100) THEN 
			IF Lynus_Standards.GVL_Energy.stDataHeatingPumps[diNrOfEMS_OUT,arrCTCheckActivePrio[2]].arrTargetPowerEMS[1] >= 100 THEN 
				arrActualStepInTurn[1] := 2; 
			ELSE 
				arrActualStepInTurn[1] := 1; 
			END_IF
			arrMaxPrioReached[2] := FALSE; 
			arrMinPrioReached[2] := FALSE;
			arrCTCheckActivePrio[2] := 0; 
			liNrOfNotDoneDevices := 0; 
			liCounterCkeckDeviceAndPrio := 0;
			uiState := 70;
		ELSE
			IF bSurplusAvailable AND arrActualPrioInTurn[2] < 255 AND uiState = 50 AND arrCTCheckActivePrio[2] = Constants_Energy.diMaxNumberOfHeatingPumps THEN 
				arrActualPrioInTurn[2] := arrActualPrioInTurn[2] + 1; 
				arrCTCheckActivePrio[2] := 0; 
				liCounterCkeckDeviceAndPrio := 0; 
				liNrOfNotDoneDevices := 0; 
			END_IF
		END_IF
		//No surplus
		IF NOT bSurplusAvailable AND Lynus_Standards.GVL_Energy.stDataHeatingPumps[diNrOfEMS_OUT,arrCTCheckActivePrio[2]].byPriority = arrActualPrioInTurn[2] AND NOT Lynus_Standards.GVL_Energy.stDataHeatingPumps[diNrOfEMS_OUT,arrCTCheckActivePrio[2]].bIsStepSwitched AND NOT 
		Lynus_Standards.GVL_Energy.stDataHeatingPumps[diNrOfEMS_OUT,arrCTCheckActivePrio[2]].bIsControllable AND Lynus_Standards.GVL_Energy.stDataHeatingPumps[diNrOfEMS_OUT,arrCTCheckActivePrio[2]].arrTargetPowerEMS[1] > 0 THEN
			arrActualStepInTurn[1] := 1;	
			arrMaxPrioReached[2] := FALSE;
			arrMinPrioReached[2] := FALSE;
			arrCTCheckActivePrio[2] := 0; 
			liNrOfNotDoneDevices := 0; 
			liCounterCkeckDeviceAndPrio := 0;
			uiState := 70;
		ELSIF NOT bSurplusAvailable AND Lynus_Standards.GVL_Energy.stDataHeatingPumps[diNrOfEMS_OUT,arrCTCheckActivePrio[2]].byPriority = arrActualPrioInTurn[2] AND Lynus_Standards.GVL_Energy.stDataHeatingPumps[diNrOfEMS_OUT,arrCTCheckActivePrio[2]].byNumberOfSteps = 0 AND 
		Lynus_Standards.GVL_Energy.stDataHeatingPumps[diNrOfEMS_OUT,arrCTCheckActivePrio[2]].arrTargetPowerEMS[1] > 0 THEN
			arrActualStepInTurn[1] := 1;	
			arrMaxPrioReached[2] := FALSE;
			arrMinPrioReached[2] := FALSE;
			arrCTCheckActivePrio[2] := 0; 
			liNrOfNotDoneDevices := 0; 
			liCounterCkeckDeviceAndPrio := 0;
			uiState := 70;
		ELSIF NOT bSurplusAvailable AND Lynus_Standards.GVL_Energy.stDataHeatingPumps[diNrOfEMS_OUT,arrCTCheckActivePrio[2]].byPriority = arrActualPrioInTurn[2] AND NOT Lynus_Standards.GVL_Energy.stDataHeatingPumps[diNrOfEMS_OUT,arrCTCheckActivePrio[2]].bIsStepSwitched AND 
		Lynus_Standards.GVL_Energy.stDataHeatingPumps[diNrOfEMS_OUT,arrCTCheckActivePrio[2]].bIsControllable AND Lynus_Standards.GVL_Energy.stDataHeatingPumps[diNrOfEMS_OUT,arrCTCheckActivePrio[2]].arrTargetPowerEMS[1] > 0 THEN
			arrActualStepInTurn[1] := 1;	
			arrMaxPrioReached[2] := FALSE;
			arrMinPrioReached[2] := FALSE;
			arrCTCheckActivePrio[2] := 0; 
			liNrOfNotDoneDevices := 0; 
			liCounterCkeckDeviceAndPrio := 0;
			uiState := 70;
		ELSIF NOT bSurplusAvailable AND Lynus_Standards.GVL_Energy.stDataHeatingPumps[diNrOfEMS_OUT,arrCTCheckActivePrio[2]].byPriority = arrActualPrioInTurn[2] AND Lynus_Standards.GVL_Energy.stDataHeatingPumps[diNrOfEMS_OUT,arrCTCheckActivePrio[2]].bIsStepSwitched AND 
		Lynus_Standards.GVL_Energy.stDataHeatingPumps[diNrOfEMS_OUT,arrCTCheckActivePrio[2]].bIsControllable AND Lynus_Standards.GVL_Energy.stDataHeatingPumps[diNrOfEMS_OUT,arrCTCheckActivePrio[2]].byNumberOfSteps = 1 AND Lynus_Standards.GVL_Energy.stDataHeatingPumps[diNrOfEMS_OUT,arrCTCheckActivePrio[2]].arrTargetPowerEMS[1] > 0 THEN
			arrActualStepInTurn[1] := 1;	
			arrMaxPrioReached[2] := FALSE;
			arrMinPrioReached[2] := FALSE;
			arrCTCheckActivePrio[2] := 0; 
			liNrOfNotDoneDevices := 0; 
			liCounterCkeckDeviceAndPrio := 0;
			uiState := 70;
		ELSIF NOT bSurplusAvailable AND Lynus_Standards.GVL_Energy.stDataHeatingPumps[diNrOfEMS_OUT,arrCTCheckActivePrio[2]].byPriority = arrActualPrioInTurn[2] AND Lynus_Standards.GVL_Energy.stDataHeatingPumps[diNrOfEMS_OUT,arrCTCheckActivePrio[2]].bIsStepSwitched AND 
		Lynus_Standards.GVL_Energy.stDataHeatingPumps[diNrOfEMS_OUT,arrCTCheckActivePrio[2]].bIsControllable AND Lynus_Standards.GVL_Energy.stDataHeatingPumps[diNrOfEMS_OUT,arrCTCheckActivePrio[2]].byNumberOfSteps = 2 AND (Lynus_Standards.GVL_Energy.stDataHeatingPumps[diNrOfEMS_OUT,arrCTCheckActivePrio[2]].arrTargetPowerEMS[1] > 0 OR Lynus_Standards.GVL_Energy.stDataHeatingPumps[diNrOfEMS_OUT,arrCTCheckActivePrio[2]].arrTargetPowerEMS[2] > 0) THEN
			IF Lynus_Standards.GVL_Energy.stDataHeatingPumps[diNrOfEMS_OUT,arrCTCheckActivePrio[2]].arrTargetPowerEMS[2] <= 0 THEN 
				arrActualStepInTurn[1] := 1; 
			ELSE 
				arrActualStepInTurn[1] := 2; 
			END_IF
			arrMaxPrioReached[2] := FALSE;
			arrMinPrioReached[2] := FALSE;	
			arrCTCheckActivePrio[2] := 0; 
			liNrOfNotDoneDevices := 0; 
			liCounterCkeckDeviceAndPrio := 0;
			uiState := 70;
		ELSE
			IF NOT bSurplusAvailable AND arrActualPrioInTurn[2] > 1 AND uiState = 50 AND arrCTCheckActivePrio[2] = Constants_Energy.diMaxNumberOfHeatingPumps THEN 
				arrActualPrioInTurn[2] := arrActualPrioInTurn[2] - 1; 
				arrCTCheckActivePrio[2] := 0; 
				liCounterCkeckDeviceAndPrio := 0;  
				liNrOfNotDoneDevices := 0; 
			END_IF
		END_IF 	  
	
		//Go to next step if we are on min prio or on max prio and the target power is just set to the min or to the max value.
		liCounterCkeckDeviceAndPrio := LIMIT(0,liCounterCkeckDeviceAndPrio,Constants_Energy.diMaxNumberOfHeatingPumps);
		
		IF arrActualPrioInTurn[2] = 1 AND Lynus_Standards.GVL_Energy.stDataHeatingPumps[diNrOfEMS_OUT,liCounterCkeckDeviceAndPrio].byPriority = 1 AND
			(Lynus_Standards.GVL_Energy.stDataHeatingPumps[diNrOfEMS_OUT,liCounterCkeckDeviceAndPrio].arrTargetPowerEMS[1] <> 0 OR Lynus_Standards.GVL_Energy.stDataHeatingPumps[diNrOfEMS_OUT,liCounterCkeckDeviceAndPrio].arrTargetPowerEMS[2] <> 0) THEN 
				liNrOfNotDoneDevices := liNrOfNotDoneDevices + 1; 
		END_IF
		//1 Step
		IF arrActualPrioInTurn[2] = 255 AND Lynus_Standards.GVL_Energy.stDataHeatingPumps[diNrOfEMS_OUT,liCounterCkeckDeviceAndPrio].byPriority = 255 AND Lynus_Standards.GVL_Energy.stDataHeatingPumps[diNrOfEMS_OUT,liCounterCkeckDeviceAndPrio].byNumberOfSteps = 1 AND  
			Lynus_Standards.GVL_Energy.stDataHeatingPumps[diNrOfEMS_OUT,liCounterCkeckDeviceAndPrio].arrTargetPowerEMS[1] < 100 THEN 
				liNrOfNotDoneDevices := liNrOfNotDoneDevices + 1; 
		//2 Steps
		ELSIF arrActualPrioInTurn[2] = 255 AND Lynus_Standards.GVL_Energy.stDataHeatingPumps[diNrOfEMS_OUT,liCounterCkeckDeviceAndPrio].byPriority = 255 AND Lynus_Standards.GVL_Energy.stDataHeatingPumps[diNrOfEMS_OUT,liCounterCkeckDeviceAndPrio].byNumberOfSteps = 2 AND  
			(Lynus_Standards.GVL_Energy.stDataHeatingPumps[diNrOfEMS_OUT,liCounterCkeckDeviceAndPrio].arrTargetPowerEMS[1] < 100 OR Lynus_Standards.GVL_Energy.stDataHeatingPumps[diNrOfEMS_OUT,liCounterCkeckDeviceAndPrio].arrTargetPowerEMS[2] < 100) THEN 
				liNrOfNotDoneDevices := liNrOfNotDoneDevices + 1; 
		END_IF
	
		
		IF arrActualPrioInTurn[2] = 1 AND uiState = 50 AND liNrOfNotDoneDevices = 0 AND arrCTCheckActivePrio[2] = Constants_Energy.diMaxNumberOfHeatingPumps AND liCounterCkeckDeviceAndPrio = Constants_Energy.diMaxNumberOfHeatingPumps THEN 
			arrMinPrioReached[2] := TRUE; arrMaxPrioReached[2] := FALSE; liNrOfNotDoneDevices := 0; uiState := 70; arrCTCheckActivePrio[2] := 0; liCounterCkeckDeviceAndPrio := 0; 
		END_IF
		IF arrActualPrioInTurn[2] = 255 AND uiState = 50 AND liNrOfNotDoneDevices = 0 AND arrCTCheckActivePrio[2] = Constants_Energy.diMaxNumberOfHeatingPumps AND  liCounterCkeckDeviceAndPrio = Constants_Energy.diMaxNumberOfHeatingPumps THEN 
			arrMaxPrioReached[2] := TRUE; arrMinPrioReached[2] := FALSE; liNrOfNotDoneDevices := 0; uiState := 70; arrCTCheckActivePrio[2] := 0; liCounterCkeckDeviceAndPrio := 0;
		END_IF
		
		//Timout, go to next step
		IF timTimeout.Q AND uiState = 50 THEN 
			uiState := 70; 
		END_IF
		
	70: //Check the priority for the electric heating element incl. the steps to controll it
		uiState_CP := uiState;
	
		//Counter to ckeck if we reached at the min or the max prio
		IF uiState = 70 THEN 
			liCounterCkeckDeviceAndPrio := liCounterCkeckDeviceAndPrio + 1; 
		END_IF
	
		//First check if we have min 1 of this Device Type. If not, complete this Device Type and go to the next step
		//Check also the bigest Priority of this Device Type
		diNumberOfDevicesFromEachType := 0; bySearchBigestPrio := 0;
		FOR liLPCheckDeviceAndPrio := 1 TO Constants_Energy.diMaxNumberOfElectricHeatingElements BY 1 DO
			IF Lynus_Standards.GVL_Energy.stDataElectricHeatingElements[diNrOfEMS_OUT,liLPCheckDeviceAndPrio].byPriority <> 0 THEN 
				diNumberOfDevicesFromEachType := diNumberOfDevicesFromEachType + 1; 
			END_IF
			IF Lynus_Standards.GVL_Energy.stDataElectricHeatingElements[diNrOfEMS_OUT,liLPCheckDeviceAndPrio].byPriority > bySearchBigestPrio THEN 
				bySearchBigestPrio := Lynus_Standards.GVL_Energy.stDataElectricHeatingElements[diNrOfEMS_OUT,liLPCheckDeviceAndPrio].byPriority; 
			END_IF   
		END_FOR 
		IF bSurplusAvailable AND arrActualPrioInTurn[3] > bySearchBigestPrio AND uiState = 70 THEN 
			arrActualPrioInTurn[3] := 255; 
		END_IF
		IF NOT bSurplusAvailable AND arrActualPrioInTurn[3] > bySearchBigestPrio AND uiState = 70 THEN 
			arrActualPrioInTurn[3] := bySearchBigestPrio; 
		END_IF
		
		IF bSurplusAvailable AND diNumberOfDevicesFromEachType = 0 THEN 
			arrActualPrioInTurn[3] := 255; 
		END_IF
		IF NOT bSurplusAvailable AND diNumberOfDevicesFromEachType = 0 THEN 
			arrActualPrioInTurn[3] := 1; 
		END_IF
		
		//Count up each Device
		arrCTCheckActivePrio[3] := arrCTCheckActivePrio[3] + 1;
		arrCTCheckActivePrio[3] := LIMIT(1,arrCTCheckActivePrio[3],Constants_Energy.diMaxNumberOfElectricHeatingElements);
		
